// TIA Portal V17 export
// export: Created 2025-07-01T09:58:21.0344057Z, ExportSetting WithDefaults, DisplayName Totally Integrated Automation Portal, DisplayVersion V17 Update 8, DisplayName TIA Portal Openness, DisplayVersion V17 Update 8, DisplayName TIA Portal Version Control Interface, DisplayVersion V17, DisplayName SINAMICS Startdrive Advanced, DisplayVersion V17 SP2, DisplayName SINAMICS Startdrive G110M, G120, G120C, G120D, G120P, G115D, DisplayVersion V17 SP2, DisplayName SINAMICS Startdrive G130, G150, S120, S150, SINAMICS MV, S210, DisplayVersion V17 SP2, DisplayName STEP 7 Professional, DisplayVersion V17 Update 8, DisplayName SINUMERIK ONE STEP 7 Toolbox, DisplayVersion V17 Update 12, DisplayName SINUMERIK ONE PLC Basic Program Plus, DisplayVersion V17 Update 12, DisplayName SINUMERIK 840D sl STEP 7 Toolbox, DisplayVersion V17 Update 12, DisplayName STEP 7 Safety, DisplayVersion V17 Update 6, DisplayName WinCC Advanced, DisplayVersion V17 Update 8
FUNCTION_BLOCK "FB31_SPINDLE"   // FB31, LAD
{ S7_Optimized_Access := 'FALSE' }
AUTHOR : ETXETAR
VERSION : 1.0
// stored: AutoNumber false, IsIECCheckEnabled false, SetENOAutomatically false, UDAEnableTagReadback false
   VAR_INPUT
      OPTIONS_0 : Byte := 2#0000_0000;   // OPTIONS 0
      OPTIONS_1 : Byte := 2#0000_0000;   // OPTIONS 1
      SAFETY_BYPASS : Bool;   // MUST BE ALWAYS OFF, ACTIVATE ONLY FOR TEST
      OPTIMIZATION_BYPASS : Bool;   // MUST BE ALWAYS OFF, ACTIVATE ONLY FOR OPTIMIZATION TEST
      RPMS_REACHED : Bool;   // RPMS REACHED / N.O
      BELT_BROKEN : Bool;   // BELT BROKEN / N.C
      COOLING_SYS_IN_SERVICE : Bool;   // COOLING SYSTEM IN SERVICE
      MQL_HP_IN_SERVICE : Bool;   // MQL OR HP IN SERVICE
      TEMPERATURE_SENSOR : Word;   // TEMPERATURE SENSOR
      TEMPERATURE_SENSOR_PTC : Bool;   // TEMPERATURE SENSOR PTC
      VPM_READY : Bool;   // VOLTAGE PROTECTION MODULE READY
      ENABLE : Bool;   // ENABLE
      FEED_HOLD_COND : Bool;   // FEED HOLD CONDITION
      UNIT_SEQ_RUNNING : Bool;   // UNIT SEQUENCE RUNNING
      SAFE_ENABLED : Bool;   // SAFETY ENABLED
      TEST_STOP_INTERNAL_PULSES : Bool;   // TEST STOP INTERNAL PULSES
      FEED_OVERRIDE : Byte;   // FEED OVERRIDE
      SPINDLE_OVERRIDE : Byte;   // SPINDLE OVERRIDE
      HMI_SP_SELECTED : Bool;   // HMI SPINDLE SELECTED
      HMI_REQ_LINE : Bool;   // HMI REQUEST LINE
      CHANNEL_M3 : Bool;   // CHANNEL M3
      CHANNEL_M300 : Bool;   // CHANNEL M300
      M_VERIFY_CLAMP_F1 : Bool;   // M VERIFY CLAMPED FIXTURE 1
      M_VERIFY_CLAMP_F2 : Bool;   // M VERIFY CLAMPED FIXTURE 2
      SP_CLAMP : Bool;   // SPINDLE CLAMPING UNIT CLAMP
      SP_CLAMPED : Bool;   // SPINDLE CLAMPING UNIT CLAMPED
      SP_CLAMPED_WITH_TOOL : Bool;   // SPINDLE CLAMPING UNIT CLAMPED WITH TOOL
      HARDWARE_ENABLE : Bool;   // HARDWARE ENABLE
      TOOL_CHANGE_POS : Bool;   // TOOL CHANGE POSITION
      FIXTURE_1_PART_OK : Bool;   // FIXTURE 1 PART OK
      FIXTURE_2_PART_OK : Bool;   // FIXTURE 2 PART OK
      READ_POS : DWord;   // READ POSITION
      UNIT_ALARM : UInt;   // UNIT NUMBER MAX. NUMBER=10
      STATION_ALARM : UInt;   // STATION NUMBER MIN. NUMBER=0 MAX. NUMBER=4
      DESELECT_SPINDLE_STO : Bool;   // DESELECT SPINDLE STO
   END_VAR
   VAR_OUTPUT
      DELAYED_ENABLE : Bool;   // DELAYED ENABLE
      FEED_HOLD_CONDITIONS : Bool;   // FEED HOLD CONDITIONS
      FEED_HOLD_CONDITIONS_HMI : Bool;   // HMI FEED HOLD CONDITIONS
      SP_DESELECTED : Bool;   // SPINDLE DESELECTED
      SPEED_NOT_REACHED_ALARM : Bool;   // SPEED NOT REACHED ALARM
      BELT_BROKEN_ALARM : Bool;   // BELT BROKEN ALARM
      COOLING_ALARM : Bool;   // COOLING ALARM
      MQL_HP_ALARM : Bool;   // MQL HP ALARM
      HIGH_TEMP_ALARM : Bool;   // HIGH TEMPERATURE ALARM
      HIGH_TEMP_PTC_ALARM : Bool;   // HIGH TEMPERATURE PTC ALARM
      VPM_READY_ALARM : Bool;   // VPM READY ALARM
      HIGH_TEMP_PREALM : Bool;   // HIGH TEMPERATURE PREALARM
      SPINDLE_POS : Real;   // SPINDLE POSITION
      HMI_MOTION_EXECUTABILITY_LEFT : Bool;   // HMI MOTION EXECUTABILITY LEFT
      HMI_MOTION_EXECUTABILITY_RIGHT : Bool;   // HMI MOTION EXECUTABILITY RIGHT
      HMI_MOTION_END_POS_LEFT : Bool;   // HMI MOTION END POSITION LEFT
      HMI_MOTION_END_POS_RIGHT : Bool;   // HMI MOTION END POSITION RIGHT
   END_VAR
   VAR_IN_OUT
      SpindleDB : "LBP_typeAxisX";
   END_VAR
   VAR DB_SPECIFIC
      SP : "SPINDLE";
      SP_TEMPERATURE : Real;   // SPINDLE TEMPERATURE
      TEMP_MUL_VAL { S7_SetPoint := 'True'} : Real := 800.0;   // CONVERSION VALUE TO MUL THE INPUT
      TEMP_DIV_VAL { S7_SetPoint := 'True'} : Real := 16383.0;   // CONVERSION VALUE TO DIV THE MUL VALUE
      TEMP_SUB_VAL { S7_SetPoint := 'True'} : Real := 200.0;   // CONVERSION VALUE TO SUB TO THE SUB VALUE
      TEMP_PREALARM_VAL { S7_SetPoint := 'True'} : Real := 40.0;   // TEMPERATURE PREALARM VALUE
      TEMP_ALARM_VAL { S7_SetPoint := 'True'} : Real := 45.0;   // TEMPERATURE ALARM VALUE
      WARNING_GONE { S7_SetPoint := 'True'} : Bool;   // WARNING GONE
      TIMER_ENABLE_PULSE { S7_SetPoint := 'True'} : TOF_TIME;   // ENABLE PULSE TIMER
      TIMER_DELETE_DIST_TO_GO { S7_SetPoint := 'True'} : TON_TIME;   // DELETE DISTANCE TO GO TIMER
      TIMER_SPEED_NOT_REACHED { S7_SetPoint := 'True'} : TOF_TIME;   // SPEED NOT REACHED TIMER
      TIMER_BELT_BROKEN_ALARM { S7_SetPoint := 'True'} : TON_TIME;   // BELT BROKEN TIMER
      TIMER_MQL_HP_FAULT { S7_SetPoint := 'True'} : TON_TIME;   // MQL OR HP FAULT TIMER
      TIMER_COMMAND_JOG_PLUS { S7_SetPoint := 'True'} : TON_TIME;   // COMMAND JOG PLUS TIMER
   END_VAR
   VAR
      SAFETY_POSITIONS { S7_SetPoint := 'True'} : "FB33_SAFETY_POSITIONS";
   END_VAR
   VAR_TEMP
      INPUTS_MASK : Byte;   // INPUT MASK
      O_BYTE_0 : Struct   // OPTION BYTE 0
         MEASURING_SYSTEM_2 : Bool;   // MEASURING SYSTEM 2 OPTION / ALWAYS ON OR ALWAYS OFF
         BELT_BROKEN : Bool;   // BELT BROKEN OPTION
         COOLING : Bool;   // COOLING OPTION / ALWAYS ON OR ALWAYS OFF
         MQL_OR_HP : Bool;   // MQL OR HP OPTION / ALWAYS ON OR ALWAYS OFF
         ANALOG_TEMPERATURE_SENSOR : Bool;   // ANALOG TEMPERATURE SENSOR OPTION
         PTC_TEMP_SENSOR : Bool;   // PTC TEMPERATURE SENSOR OPTION
         TWIN_KESSLER_VPM_READY : Bool;   // TWIN KESSLER VPM READY OPTION
         MPP_SP_OVERRIDE : Bool;   // MPP SPINDLE OVERRIDE OPTION
      END_STRUCT;
      O_BYTE_1 : Struct   // OPTION BYTE 1
         SPARE_0 : Bool;   // SPARE OPTION / ALWAYS ON OR ALWAYS OFF
         SPARE_1 : Bool;   // SPARE OPTION
         SPARE_2 : Bool;   // SPARE OPTION / ALWAYS ON OR ALWAYS OFF
         SPARE_3 : Bool;   // SPARE OPTION / ALWAYS ON OR ALWAYS OFF
         SPARE_4 : Bool;   // SPARE OPTION
         SPARE_5 : Bool;   // SPARE OPTION
         SPARE_6 : Bool;   // SPARE OPTION
         SPARE_7 : Bool;   // SPARE OPTION
      END_STRUCT;
      TEMP_INPUT : DInt;   // TEMPERATURE INPUR SHIFTED
      TEMP_REAL : Real;   // TEMPERATURE IN REAL
      DB_NUMBER : DInt;   // DB NUMBER FOR ALARMS AND HELP DECODING
   END_VAR
   // TIMER_ENABLE_PULSE.PT := T#1s;
   // TIMER_DELETE_DIST_TO_GO.PT := T#20ms;
   // TIMER_SPEED_NOT_REACHED.PT := T#100ms;
   // TIMER_BELT_BROKEN_ALARM.PT := T#150ms;
   // TIMER_MQL_HP_FAULT.PT := T#50ms;
   // TIMER_COMMAND_JOG_PLUS.PT := T#100ms;
   VAR_TEMP   // added for the SCL form of the ladder/FBD networks
      _w1 : Bool;
      _w2 : Bool;
      _w3 : Bool;
      _w4 : Bool;
      _w5 : Bool;
      _w6 : Bool;
      _w7 : Bool;
      _w8 : Bool;
      _w9 : Bool;
      _w10 : Bool;
      _w11 : Bool;
   END_VAR
BEGIN

NETWORK
TITLE = READ INSTANCE DB
      L     DINO;
      +     10#800000;
      T     #DB_NUMBER;


REGION Network 2: OPTIONS
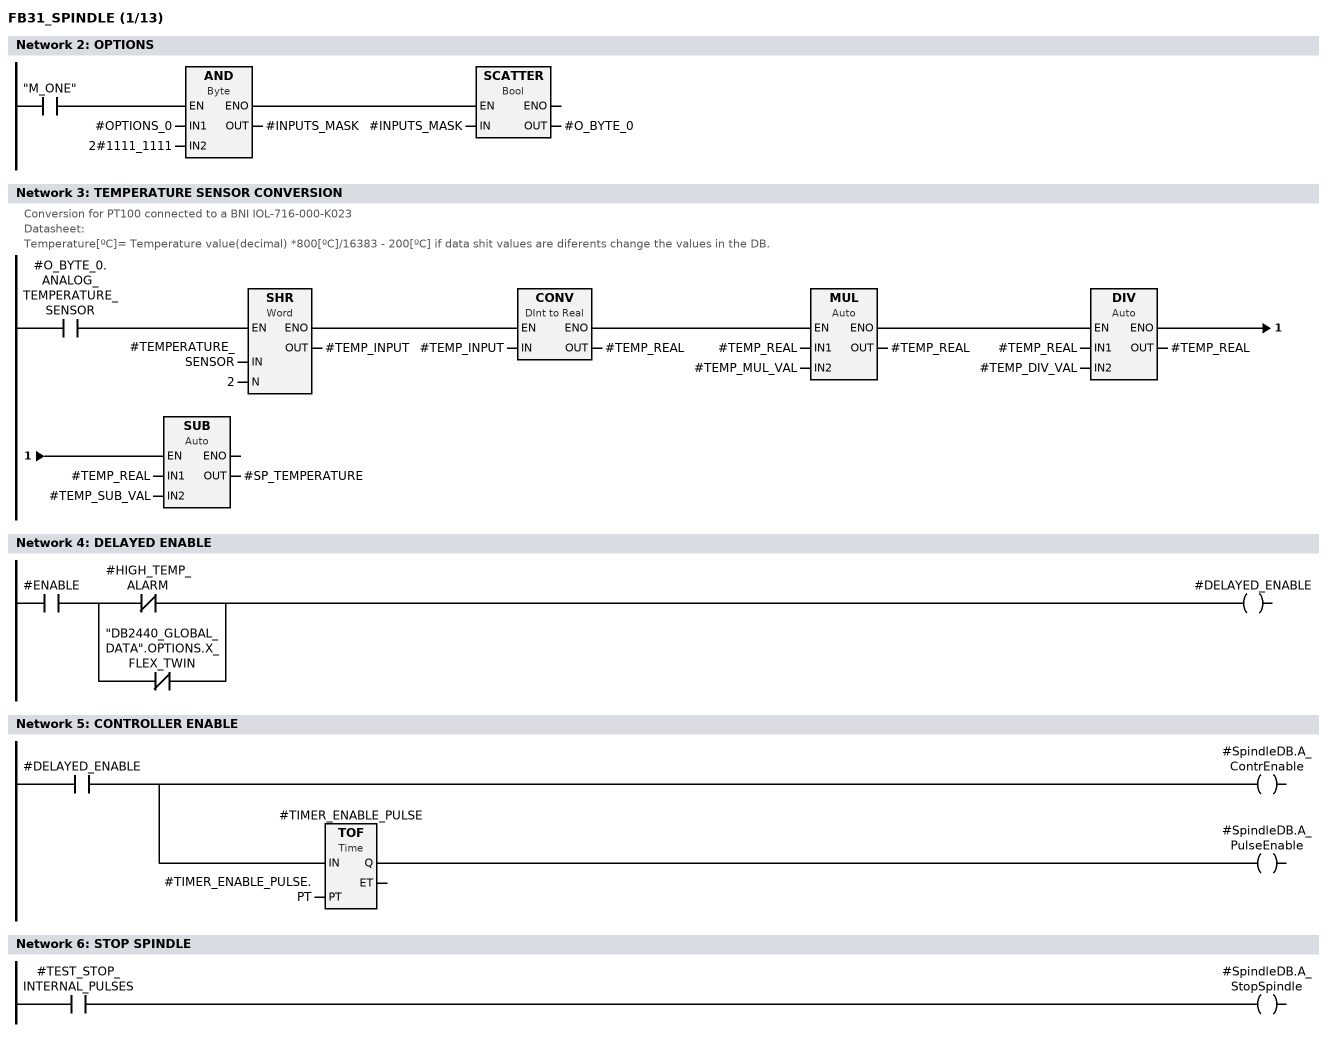
   RUNG wire#powerrail
      Contact( "M_ONE" )
      { S7_Templates := "SrcType := Byte"; S7_GenerateENO := "TRUE" } And(in1 := #OPTIONS_0, in2 := 2#1111_1111, out => #INPUTS_MASK)
      { S7_Templates := "[dest_type := Bool, src_type := Byte]" } SCATTER(IN := #INPUTS_MASK, OUT => #O_BYTE_0)
   END_RUNG
   // the same network as SCL:
   IF "M_ONE" THEN
       #INPUTS_MASK := #OPTIONS_0 AND 2#1111_1111;
       SCATTER(IN := #INPUTS_MASK, OUT => #O_BYTE_0);
   END_IF;
END_REGION

REGION Network 3: TEMPERATURE SENSOR CONVERSION
   // Conversion for PT100 connected to a BNI IOL-716-000-K023
   // 
   // Datasheet:
   // 
   //  Temperature[ºC]= Temperature value(decimal) *800[ºC]/16383 - 200[ºC] if data shit values are diferents change the values in the DB.
   RUNG wire#powerrail
      Contact( #O_BYTE_0.ANALOG_TEMPERATURE_SENSOR )
      { S7_Templates := "SrcType := Word" } Shr(in := #TEMPERATURE_SENSOR, n := 2, out => #TEMP_INPUT)
      { S7_Templates := "[SrcType := DInt, DestType := Real]" } Convert(in := #TEMP_INPUT, out => #TEMP_REAL)
      Mul(in1 := #TEMP_REAL, in2 := #TEMP_MUL_VAL, out => #TEMP_REAL)
      Div(in1 := #TEMP_REAL, in2 := #TEMP_DIV_VAL, out => #TEMP_REAL)
      Sub(in1 := #TEMP_REAL, in2 := #TEMP_SUB_VAL, out => #SP_TEMPERATURE)
   END_RUNG
   // the same network as SCL:
   IF #O_BYTE_0.ANALOG_TEMPERATURE_SENSOR THEN
       #TEMP_INPUT := SHR(IN := #TEMPERATURE_SENSOR, N := 2);
       #TEMP_REAL := DINT_TO_REAL(#TEMP_INPUT);
       #TEMP_REAL := #TEMP_REAL * #TEMP_MUL_VAL;
       #TEMP_REAL := #TEMP_REAL / #TEMP_DIV_VAL;
       #SP_TEMPERATURE := #TEMP_REAL - #TEMP_SUB_VAL;
   END_IF;
END_REGION

REGION Network 4: DELAYED ENABLE
   RUNG wire#powerrail
      Contact( #ENABLE )
      wire#w1
      I_Contact( #HIGH_TEMP_ALARM )
      wire#w2
      Coil( #DELAYED_ENABLE )
   END_RUNG
   RUNG wire#w1
      I_Contact( "DB2440_GLOBAL_DATA".OPTIONS.X_FLEX_TWIN )
   END_RUNG wire#w2
   // the same network as SCL:
   #DELAYED_ENABLE := #ENABLE AND (NOT #HIGH_TEMP_ALARM OR NOT "DB2440_GLOBAL_DATA".OPTIONS.X_FLEX_TWIN);
END_REGION

REGION Network 5: CONTROLLER ENABLE
   RUNG wire#powerrail
      Contact( #DELAYED_ENABLE )
      wire#w1
      Coil( #SpindleDB.A_ContrEnable )
   END_RUNG
   RUNG wire#w1
      { S7_Templates := "time_type := Time" } #TIMER_ENABLE_PULSE.TOF(pt := #TIMER_ENABLE_PULSE.PT, et =>)
      Coil( #SpindleDB.A_PulseEnable )
   END_RUNG
   // the same network as SCL:
   #SpindleDB.A_ContrEnable := #DELAYED_ENABLE;
   #TIMER_ENABLE_PULSE(IN := #DELAYED_ENABLE, PT := #TIMER_ENABLE_PULSE.PT);   // TOF
   #SpindleDB.A_PulseEnable := #TIMER_ENABLE_PULSE.Q;
END_REGION

REGION Network 6: STOP SPINDLE
   RUNG wire#powerrail
      Contact( #TEST_STOP_INTERNAL_PULSES )
      Coil( #SpindleDB.A_StopSpindle )
   END_RUNG
   // the same network as SCL:
   #SpindleDB.A_StopSpindle := #TEST_STOP_INTERNAL_PULSES;
END_REGION

REGION Network 7: DELETE DISTANCE TO GO / DELETE S VALUE
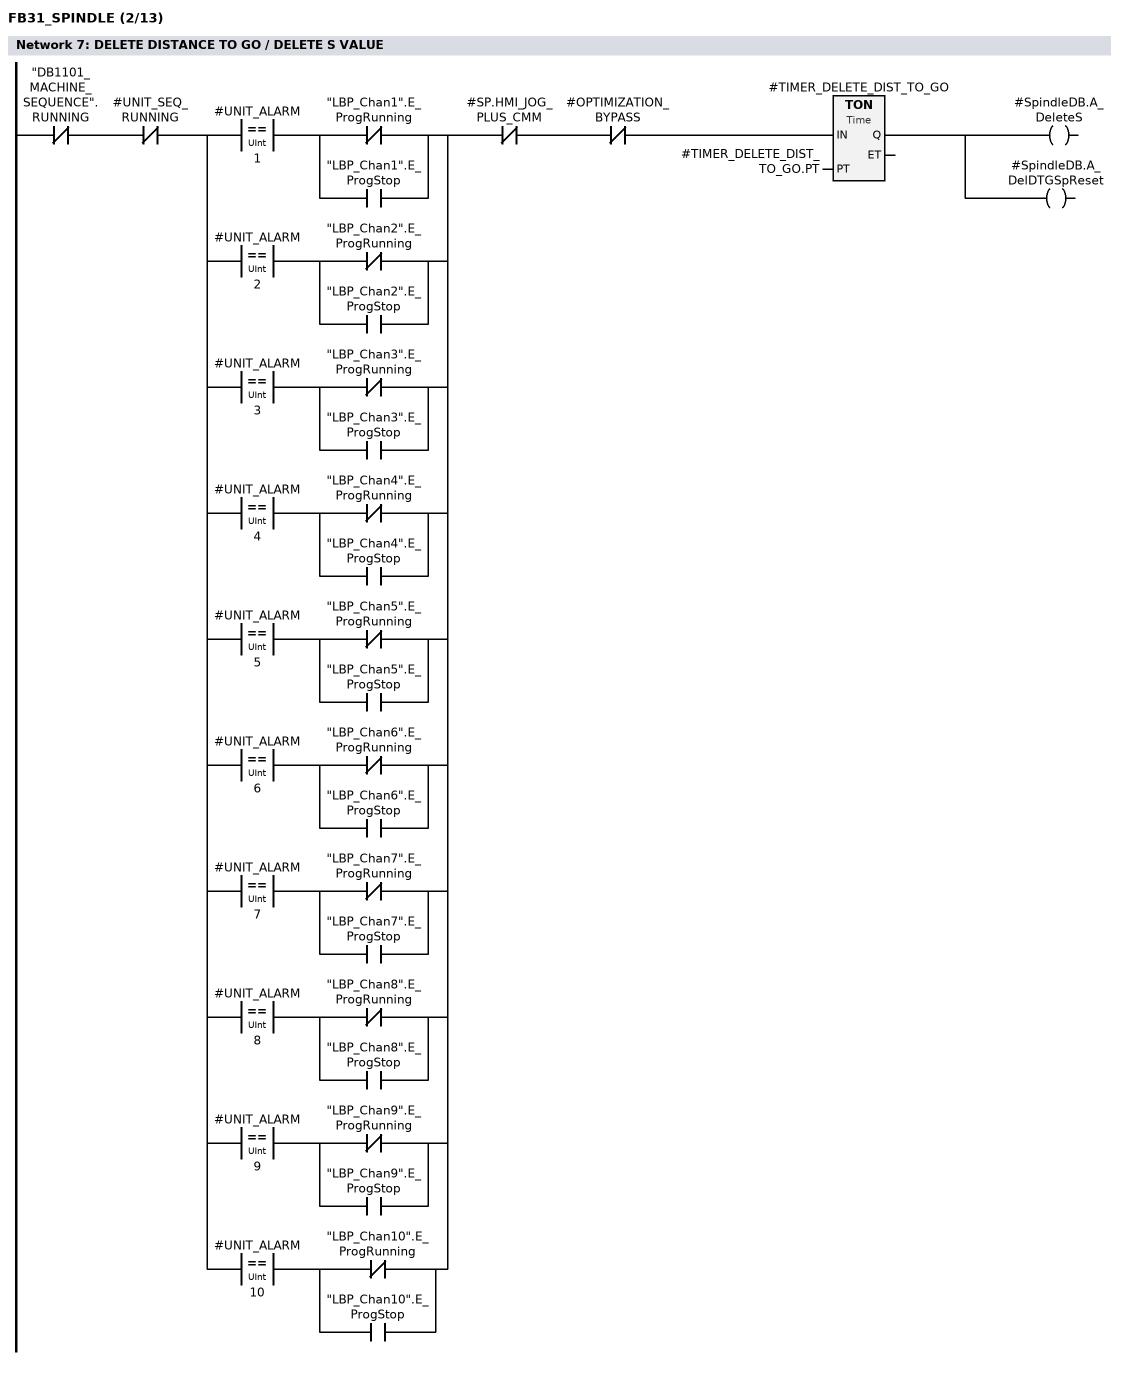
   RUNG wire#powerrail
      I_Contact( "DB1101_MACHINE_SEQUENCE".RUNNING )
      I_Contact( #UNIT_SEQ_RUNNING )
      wire#w1
      { S7_Templates := "SrcType := UInt" } EQ_Contact(in1 := #UNIT_ALARM, in2 := 1)
      wire#w2
      I_Contact( "LBP_Chan1".E_ProgRunning )
      wire#w3
      I_Contact( #SP.HMI_JOG_PLUS_CMM )
      I_Contact( #OPTIMIZATION_BYPASS )
      { S7_Templates := "time_type := Time" } #TIMER_DELETE_DIST_TO_GO.TON(pt := #TIMER_DELETE_DIST_TO_GO.PT, et =>)
      wire#w13
      Coil( #SpindleDB.A_DeleteS )
   END_RUNG
   RUNG wire#w2
      Contact( "LBP_Chan1".E_ProgStop )
   END_RUNG wire#w3
   RUNG wire#w1
      { S7_Templates := "SrcType := UInt" } EQ_Contact(in1 := #UNIT_ALARM, in2 := 2)
      wire#w4
      I_Contact( "LBP_Chan2".E_ProgRunning )
   END_RUNG wire#w3
   RUNG wire#w4
      Contact( "LBP_Chan2".E_ProgStop )
   END_RUNG wire#w3
   RUNG wire#w1
      { S7_Templates := "SrcType := UInt" } EQ_Contact(in1 := #UNIT_ALARM, in2 := 3)
      wire#w5
      I_Contact( "LBP_Chan3".E_ProgRunning )
   END_RUNG wire#w3
   RUNG wire#w5
      Contact( "LBP_Chan3".E_ProgStop )
   END_RUNG wire#w3
   RUNG wire#w1
      { S7_Templates := "SrcType := UInt" } EQ_Contact(in1 := #UNIT_ALARM, in2 := 4)
      wire#w6
      I_Contact( "LBP_Chan4".E_ProgRunning )
   END_RUNG wire#w3
   RUNG wire#w6
      Contact( "LBP_Chan4".E_ProgStop )
   END_RUNG wire#w3
   RUNG wire#w1
      { S7_Templates := "SrcType := UInt" } EQ_Contact(in1 := #UNIT_ALARM, in2 := 5)
      wire#w7
      I_Contact( "LBP_Chan5".E_ProgRunning )
   END_RUNG wire#w3
   RUNG wire#w7
      Contact( "LBP_Chan5".E_ProgStop )
   END_RUNG wire#w3
   RUNG wire#w1
      { S7_Templates := "SrcType := UInt" } EQ_Contact(in1 := #UNIT_ALARM, in2 := 6)
      wire#w8
      I_Contact( "LBP_Chan6".E_ProgRunning )
   END_RUNG wire#w3
   RUNG wire#w8
      Contact( "LBP_Chan6".E_ProgStop )
   END_RUNG wire#w3
   RUNG wire#w1
      { S7_Templates := "SrcType := UInt" } EQ_Contact(in1 := #UNIT_ALARM, in2 := 7)
      wire#w9
      I_Contact( "LBP_Chan7".E_ProgRunning )
   END_RUNG wire#w3
   RUNG wire#w9
      Contact( "LBP_Chan7".E_ProgStop )
   END_RUNG wire#w3
   RUNG wire#w1
      { S7_Templates := "SrcType := UInt" } EQ_Contact(in1 := #UNIT_ALARM, in2 := 8)
      wire#w10
      I_Contact( "LBP_Chan8".E_ProgRunning )
   END_RUNG wire#w3
   RUNG wire#w10
      Contact( "LBP_Chan8".E_ProgStop )
   END_RUNG wire#w3
   RUNG wire#w1
      { S7_Templates := "SrcType := UInt" } EQ_Contact(in1 := #UNIT_ALARM, in2 := 9)
      wire#w11
      I_Contact( "LBP_Chan9".E_ProgRunning )
   END_RUNG wire#w3
   RUNG wire#w11
      Contact( "LBP_Chan9".E_ProgStop )
   END_RUNG wire#w3
   RUNG wire#w1
      { S7_Templates := "SrcType := UInt" } EQ_Contact(in1 := #UNIT_ALARM, in2 := 10)
      wire#w12
      I_Contact( "LBP_Chan10".E_ProgRunning )
   END_RUNG wire#w3
   RUNG wire#w12
      Contact( "LBP_Chan10".E_ProgStop )
   END_RUNG wire#w3
   RUNG wire#w13
      Coil( #SpindleDB.A_DelDTGSpReset )
   END_RUNG
   // the same network as SCL:
   #TIMER_DELETE_DIST_TO_GO(IN := NOT "DB1101_MACHINE_SEQUENCE".RUNNING AND NOT #UNIT_SEQ_RUNNING AND (((#UNIT_ALARM = 1) AND (NOT "LBP_Chan1".E_ProgRunning OR "LBP_Chan1".E_ProgStop)) OR ((#UNIT_ALARM = 2) AND (NOT "LBP_Chan2".E_ProgRunning OR "LBP_Chan2".E_ProgStop)) OR ((#UNIT_ALARM = 3) AND (NOT "LBP_Chan3".E_ProgRunning OR "LBP_Chan3".E_ProgStop)) OR ((#UNIT_ALARM = 4) AND (NOT "LBP_Chan4".E_ProgRunning OR "LBP_Chan4".E_ProgStop)) OR ((#UNIT_ALARM = 5) AND (NOT "LBP_Chan5".E_ProgRunning OR "LBP_Chan5".E_ProgStop)) OR ((#UNIT_ALARM = 6) AND (NOT "LBP_Chan6".E_ProgRunning OR "LBP_Chan6".E_ProgStop)) OR ((#UNIT_ALARM = 7) AND (NOT "LBP_Chan7".E_ProgRunning OR "LBP_Chan7".E_ProgStop)) OR ((#UNIT_ALARM = 8) AND (NOT "LBP_Chan8".E_ProgRunning OR "LBP_Chan8".E_ProgStop)) OR ((#UNIT_ALARM = 9) AND (NOT "LBP_Chan9".E_ProgRunning OR "LBP_Chan9".E_ProgStop)) OR ((#UNIT_ALARM = 10) AND (NOT "LBP_Chan10".E_ProgRunning OR "LBP_Chan10".E_ProgStop))) AND NOT #SP.HMI_JOG_PLUS_CMM AND NOT #OPTIMIZATION_BYPASS,   // TON
                           PT := #TIMER_DELETE_DIST_TO_GO.PT);
   #SpindleDB.A_DeleteS := #TIMER_DELETE_DIST_TO_GO.Q;
   #SpindleDB.A_DelDTGSpReset := #TIMER_DELETE_DIST_TO_GO.Q;
END_REGION

REGION Network 8: POSITION MEASURING SYTEM
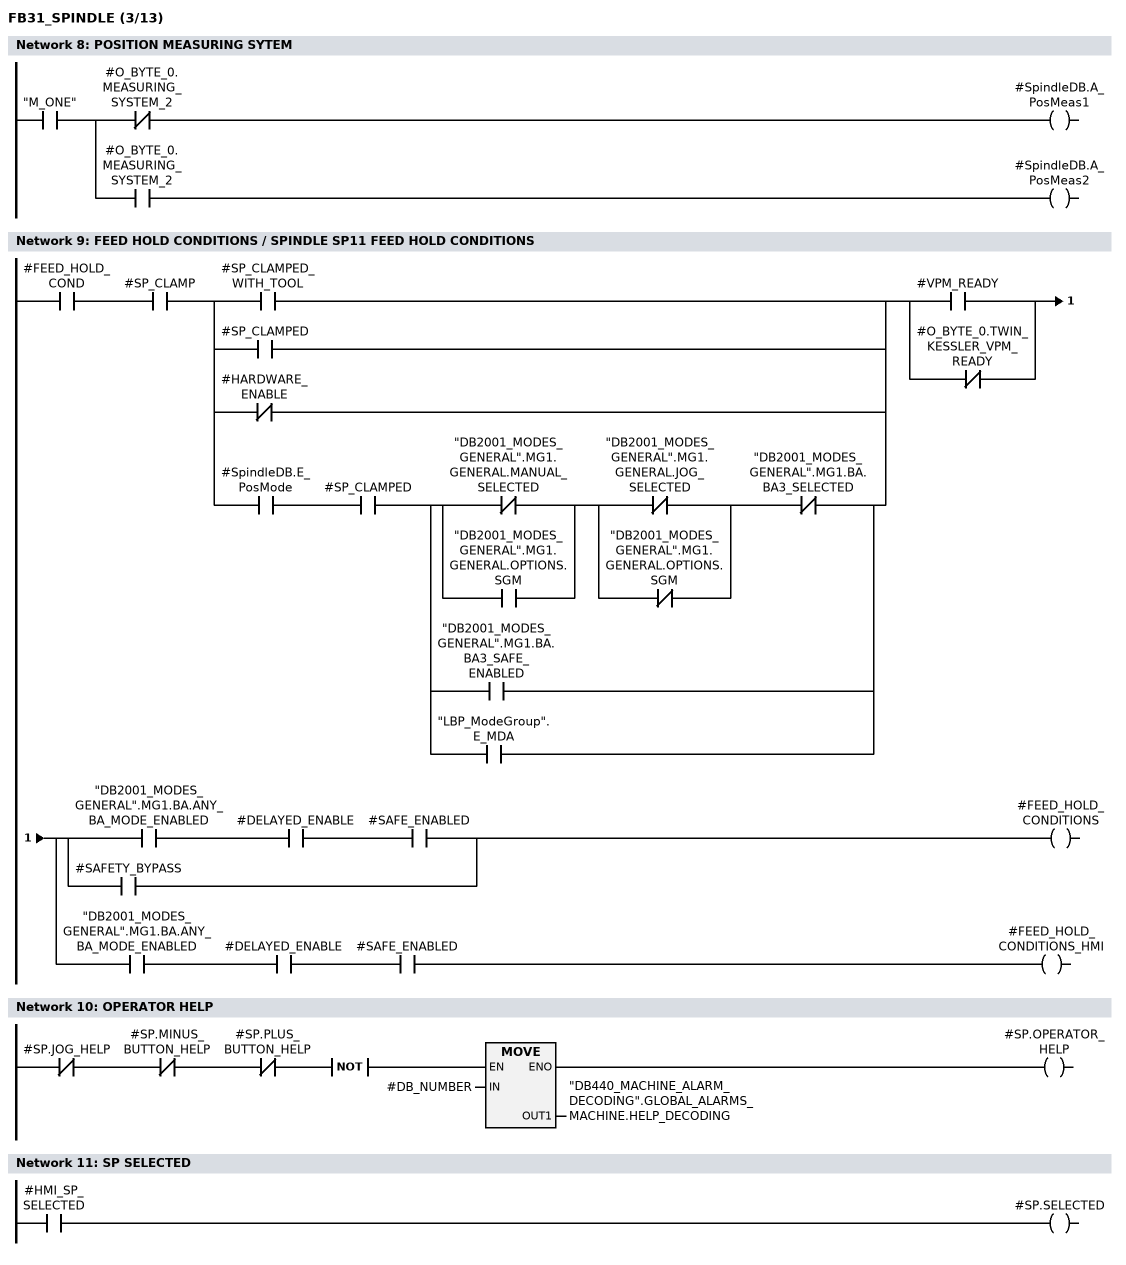
   RUNG wire#powerrail
      Contact( "M_ONE" )
      wire#w1
      I_Contact( #O_BYTE_0.MEASURING_SYSTEM_2 )
      Coil( #SpindleDB.A_PosMeas1 )
   END_RUNG
   RUNG wire#w1
      Contact( #O_BYTE_0.MEASURING_SYSTEM_2 )
      Coil( #SpindleDB.A_PosMeas2 )
   END_RUNG
   // the same network as SCL:
   #SpindleDB.A_PosMeas1 := "M_ONE" AND NOT #O_BYTE_0.MEASURING_SYSTEM_2;
   #SpindleDB.A_PosMeas2 := "M_ONE" AND #O_BYTE_0.MEASURING_SYSTEM_2;
END_REGION

REGION Network 9: FEED HOLD CONDITIONS / SPINDLE SP11 FEED HOLD CONDITIONS
   RUNG wire#powerrail
      Contact( #FEED_HOLD_COND )
      Contact( #SP_CLAMP )
      wire#w1
      Contact( #SP_CLAMPED_WITH_TOOL )
      wire#w2
      Contact( #VPM_READY )
      wire#w6
      Contact( "DB2001_MODES_GENERAL".MG1.BA.ANY_BA_MODE_ENABLED )
      Contact( #DELAYED_ENABLE )
      Contact( #SAFE_ENABLED )
      wire#w7
      Coil( #FEED_HOLD_CONDITIONS )
   END_RUNG
   RUNG wire#w1
      Contact( #SP_CLAMPED )
   END_RUNG wire#w2
   RUNG wire#w1
      I_Contact( #HARDWARE_ENABLE )
   END_RUNG wire#w2
   RUNG wire#w1
      Contact( #SpindleDB.E_PosMode )
      Contact( #SP_CLAMPED )
      wire#w3
      I_Contact( "DB2001_MODES_GENERAL".MG1.GENERAL.MANUAL_SELECTED )
      wire#w4
      I_Contact( "DB2001_MODES_GENERAL".MG1.GENERAL.JOG_SELECTED )
      wire#w5
      I_Contact( "DB2001_MODES_GENERAL".MG1.BA.BA3_SELECTED )
   END_RUNG wire#w2
   RUNG wire#w3
      Contact( "DB2001_MODES_GENERAL".MG1.GENERAL.OPTIONS.SGM )
   END_RUNG wire#w4
   RUNG wire#w4
      I_Contact( "DB2001_MODES_GENERAL".MG1.GENERAL.OPTIONS.SGM )
   END_RUNG wire#w5
   RUNG wire#w3
      Contact( "DB2001_MODES_GENERAL".MG1.BA.BA3_SAFE_ENABLED )
   END_RUNG wire#w2
   RUNG wire#w3
      Contact( "LBP_ModeGroup".E_MDA )
   END_RUNG wire#w2
   RUNG wire#w2
      I_Contact( #O_BYTE_0.TWIN_KESSLER_VPM_READY )
   END_RUNG wire#w6
   RUNG wire#w6
      Contact( #SAFETY_BYPASS )
   END_RUNG wire#w7
   RUNG wire#w6
      Contact( "DB2001_MODES_GENERAL".MG1.BA.ANY_BA_MODE_ENABLED )
      Contact( #DELAYED_ENABLE )
      Contact( #SAFE_ENABLED )
      Coil( #FEED_HOLD_CONDITIONS_HMI )
   END_RUNG
   // the same network as SCL:
   #_w1 := #FEED_HOLD_COND AND #SP_CLAMP AND (#SP_CLAMPED_WITH_TOOL OR #SP_CLAMPED OR NOT #HARDWARE_ENABLE OR (#SpindleDB.E_PosMode AND #SP_CLAMPED AND (((NOT "DB2001_MODES_GENERAL".MG1.GENERAL.MANUAL_SELECTED OR "DB2001_MODES_GENERAL".MG1.GENERAL.OPTIONS.SGM) AND (NOT "DB2001_MODES_GENERAL".MG1.GENERAL.JOG_SELECTED OR NOT "DB2001_MODES_GENERAL".MG1.GENERAL.OPTIONS.SGM) AND NOT "DB2001_MODES_GENERAL".MG1.BA.BA3_SELECTED) OR "DB2001_MODES_GENERAL".MG1.BA.BA3_SAFE_ENABLED OR "LBP_ModeGroup".E_MDA))) AND (#VPM_READY OR NOT #O_BYTE_0.TWIN_KESSLER_VPM_READY);
   #FEED_HOLD_CONDITIONS := #_w1 AND (("DB2001_MODES_GENERAL".MG1.BA.ANY_BA_MODE_ENABLED AND #DELAYED_ENABLE AND #SAFE_ENABLED) OR #SAFETY_BYPASS);
   #FEED_HOLD_CONDITIONS_HMI := #_w1 AND "DB2001_MODES_GENERAL".MG1.BA.ANY_BA_MODE_ENABLED AND #DELAYED_ENABLE AND #SAFE_ENABLED;
END_REGION

REGION Network 10: OPERATOR HELP
   RUNG wire#powerrail
      I_Contact( #SP.JOG_HELP )
      I_Contact( #SP.MINUS_BUTTON_HELP )
      I_Contact( #SP.PLUS_BUTTON_HELP )
      Not()
      { S7_GenerateENO := "TRUE" } Move(in := #DB_NUMBER, out1 => "DB440_MACHINE_ALARM_DECODING".GLOBAL_ALARMS_MACHINE.HELP_DECODING)
      Coil( #SP.OPERATOR_HELP )
   END_RUNG
   // the same network as SCL:
   // ENO of a box is taken as its EN; it also drops when the box reports an error
   #_w1 := NOT (NOT #SP.JOG_HELP AND NOT #SP.MINUS_BUTTON_HELP AND NOT #SP.PLUS_BUTTON_HELP);
   IF #_w1 THEN "DB440_MACHINE_ALARM_DECODING".GLOBAL_ALARMS_MACHINE.HELP_DECODING := #DB_NUMBER; END_IF;
   #SP.OPERATOR_HELP := #_w1;
END_REGION

REGION Network 11: SP SELECTED
   RUNG wire#powerrail
      Contact( #HMI_SP_SELECTED )
      Coil( #SP.SELECTED )
   END_RUNG
   // the same network as SCL:
   #SP.SELECTED := #HMI_SP_SELECTED;
END_REGION

REGION Network 12: SP DESELECTED
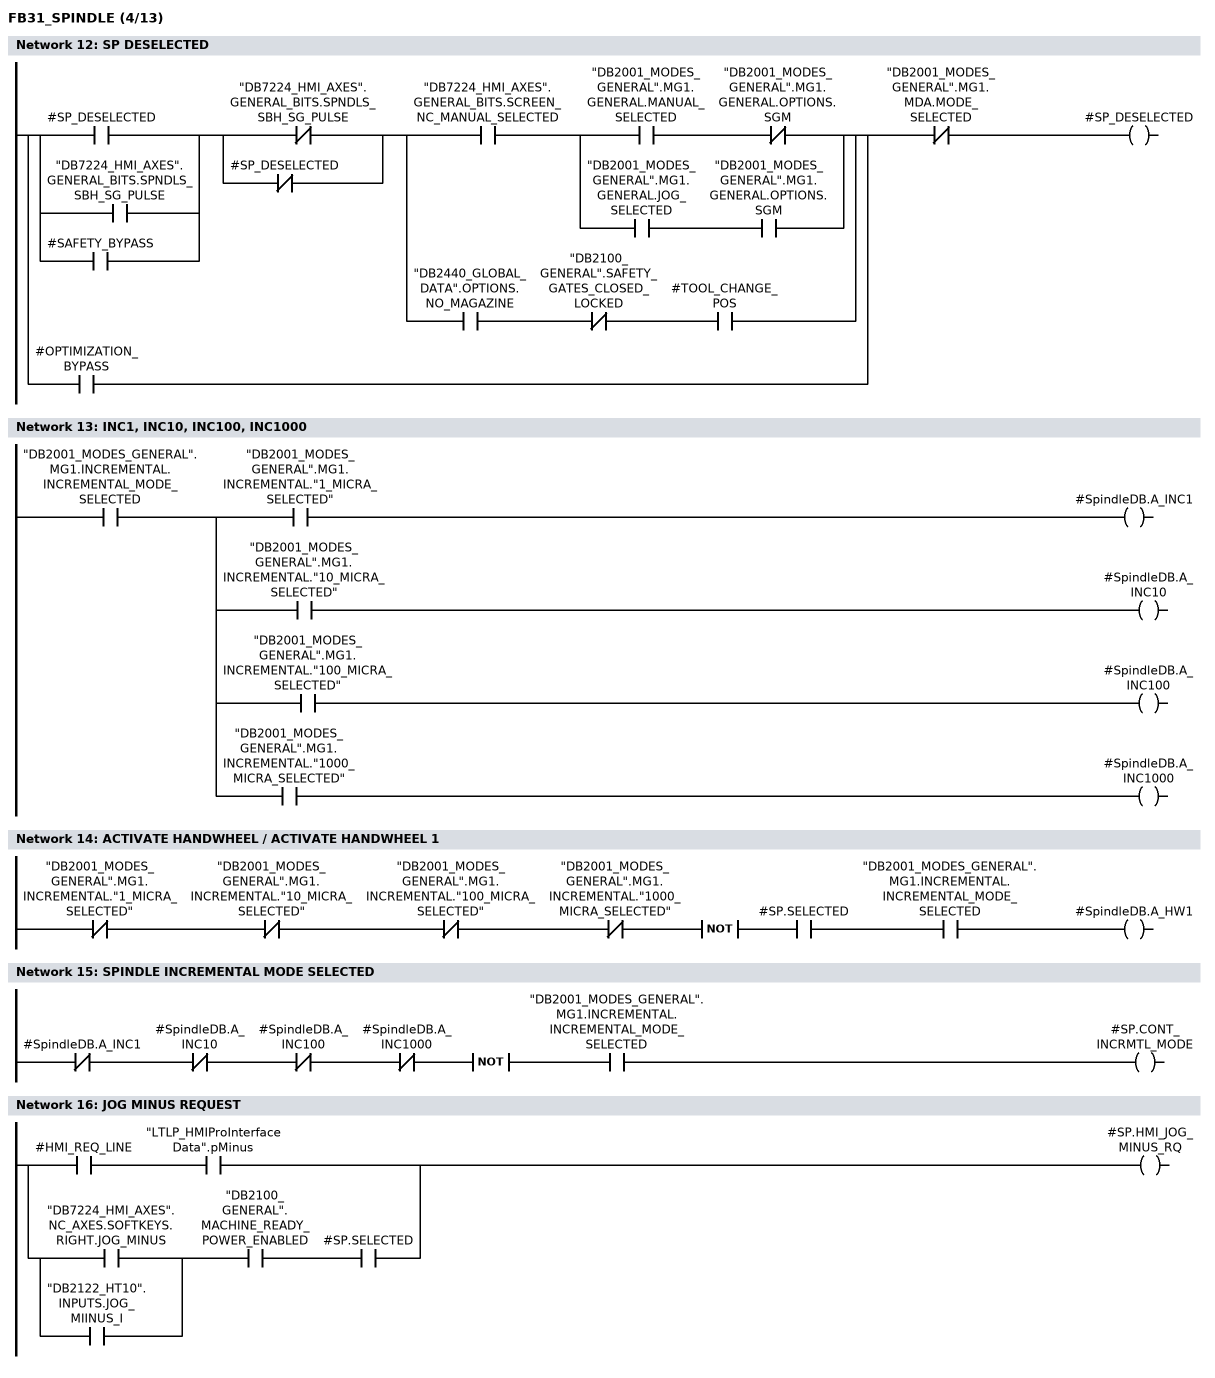
   RUNG wire#powerrail
      Contact( #SP_DESELECTED )
      wire#w1
      I_Contact( "DB7224_HMI_AXES".GENERAL_BITS.SPNDLS_SBH_SG_PULSE )
      wire#w2
      Contact( "DB7224_HMI_AXES".GENERAL_BITS.SCREEN_NC_MANUAL_SELECTED )
      wire#w3
      Contact( "DB2001_MODES_GENERAL".MG1.GENERAL.MANUAL_SELECTED )
      I_Contact( "DB2001_MODES_GENERAL".MG1.GENERAL.OPTIONS.SGM )
      wire#w4
      I_Contact( "DB2001_MODES_GENERAL".MG1.MDA.MODE_SELECTED )
      Coil( #SP_DESELECTED )
   END_RUNG
   RUNG wire#powerrail
      Contact( "DB7224_HMI_AXES".GENERAL_BITS.SPNDLS_SBH_SG_PULSE )
   END_RUNG wire#w1
   RUNG wire#powerrail
      Contact( #SAFETY_BYPASS )
   END_RUNG wire#w1
   RUNG wire#w1
      I_Contact( #SP_DESELECTED )
   END_RUNG wire#w2
   RUNG wire#w3
      Contact( "DB2001_MODES_GENERAL".MG1.GENERAL.JOG_SELECTED )
      Contact( "DB2001_MODES_GENERAL".MG1.GENERAL.OPTIONS.SGM )
   END_RUNG wire#w4
   RUNG wire#w2
      Contact( "DB2440_GLOBAL_DATA".OPTIONS.NO_MAGAZINE )
      I_Contact( "DB2100_GENERAL".SAFETY_GATES_CLOSED_LOCKED )
      Contact( #TOOL_CHANGE_POS )
   END_RUNG wire#w4
   RUNG wire#powerrail
      Contact( #OPTIMIZATION_BYPASS )
   END_RUNG wire#w4
   // the same network as SCL:
   #SP_DESELECTED := (((#SP_DESELECTED OR "DB7224_HMI_AXES".GENERAL_BITS.SPNDLS_SBH_SG_PULSE OR #SAFETY_BYPASS) AND (NOT "DB7224_HMI_AXES".GENERAL_BITS.SPNDLS_SBH_SG_PULSE OR NOT #SP_DESELECTED) AND (("DB7224_HMI_AXES".GENERAL_BITS.SCREEN_NC_MANUAL_SELECTED AND (("DB2001_MODES_GENERAL".MG1.GENERAL.MANUAL_SELECTED AND NOT "DB2001_MODES_GENERAL".MG1.GENERAL.OPTIONS.SGM) OR ("DB2001_MODES_GENERAL".MG1.GENERAL.JOG_SELECTED AND "DB2001_MODES_GENERAL".MG1.GENERAL.OPTIONS.SGM))) OR ("DB2440_GLOBAL_DATA".OPTIONS.NO_MAGAZINE AND NOT "DB2100_GENERAL".SAFETY_GATES_CLOSED_LOCKED AND #TOOL_CHANGE_POS))) OR #OPTIMIZATION_BYPASS) AND NOT "DB2001_MODES_GENERAL".MG1.MDA.MODE_SELECTED;
END_REGION

REGION Network 13: INC1, INC10, INC100, INC1000
   RUNG wire#powerrail
      Contact( "DB2001_MODES_GENERAL".MG1.INCREMENTAL.INCREMENTAL_MODE_SELECTED )
      wire#w1
      Contact( "DB2001_MODES_GENERAL".MG1.INCREMENTAL."1_MICRA_SELECTED" )
      Coil( #SpindleDB.A_INC1 )
   END_RUNG
   RUNG wire#w1
      Contact( "DB2001_MODES_GENERAL".MG1.INCREMENTAL."10_MICRA_SELECTED" )
      Coil( #SpindleDB.A_INC10 )
   END_RUNG
   RUNG wire#w1
      Contact( "DB2001_MODES_GENERAL".MG1.INCREMENTAL."100_MICRA_SELECTED" )
      Coil( #SpindleDB.A_INC100 )
   END_RUNG
   RUNG wire#w1
      Contact( "DB2001_MODES_GENERAL".MG1.INCREMENTAL."1000_MICRA_SELECTED" )
      Coil( #SpindleDB.A_INC1000 )
   END_RUNG
   // the same network as SCL:
   #SpindleDB.A_INC1 := "DB2001_MODES_GENERAL".MG1.INCREMENTAL.INCREMENTAL_MODE_SELECTED AND "DB2001_MODES_GENERAL".MG1.INCREMENTAL."1_MICRA_SELECTED";
   #SpindleDB.A_INC10 := "DB2001_MODES_GENERAL".MG1.INCREMENTAL.INCREMENTAL_MODE_SELECTED AND "DB2001_MODES_GENERAL".MG1.INCREMENTAL."10_MICRA_SELECTED";
   #SpindleDB.A_INC100 := "DB2001_MODES_GENERAL".MG1.INCREMENTAL.INCREMENTAL_MODE_SELECTED AND "DB2001_MODES_GENERAL".MG1.INCREMENTAL."100_MICRA_SELECTED";
   #SpindleDB.A_INC1000 := "DB2001_MODES_GENERAL".MG1.INCREMENTAL.INCREMENTAL_MODE_SELECTED AND "DB2001_MODES_GENERAL".MG1.INCREMENTAL."1000_MICRA_SELECTED";
END_REGION

REGION Network 14: ACTIVATE HANDWHEEL / ACTIVATE HANDWHEEL 1
   RUNG wire#powerrail
      I_Contact( "DB2001_MODES_GENERAL".MG1.INCREMENTAL."1_MICRA_SELECTED" )
      I_Contact( "DB2001_MODES_GENERAL".MG1.INCREMENTAL."10_MICRA_SELECTED" )
      I_Contact( "DB2001_MODES_GENERAL".MG1.INCREMENTAL."100_MICRA_SELECTED" )
      I_Contact( "DB2001_MODES_GENERAL".MG1.INCREMENTAL."1000_MICRA_SELECTED" )
      Not()
      Contact( #SP.SELECTED )
      Contact( "DB2001_MODES_GENERAL".MG1.INCREMENTAL.INCREMENTAL_MODE_SELECTED )
      Coil( #SpindleDB.A_HW1 )
   END_RUNG
   // the same network as SCL:
   #SpindleDB.A_HW1 := NOT (NOT "DB2001_MODES_GENERAL".MG1.INCREMENTAL."1_MICRA_SELECTED" AND NOT "DB2001_MODES_GENERAL".MG1.INCREMENTAL."10_MICRA_SELECTED" AND NOT "DB2001_MODES_GENERAL".MG1.INCREMENTAL."100_MICRA_SELECTED" AND NOT "DB2001_MODES_GENERAL".MG1.INCREMENTAL."1000_MICRA_SELECTED") AND #SP.SELECTED AND "DB2001_MODES_GENERAL".MG1.INCREMENTAL.INCREMENTAL_MODE_SELECTED;
END_REGION

REGION Network 15: SPINDLE INCREMENTAL MODE SELECTED
   RUNG wire#powerrail
      I_Contact( #SpindleDB.A_INC1 )
      I_Contact( #SpindleDB.A_INC10 )
      I_Contact( #SpindleDB.A_INC100 )
      I_Contact( #SpindleDB.A_INC1000 )
      Not()
      Contact( "DB2001_MODES_GENERAL".MG1.INCREMENTAL.INCREMENTAL_MODE_SELECTED )
      Coil( #SP.CONT_INCRMTL_MODE )
   END_RUNG
   // the same network as SCL:
   #SP.CONT_INCRMTL_MODE := NOT (NOT #SpindleDB.A_INC1 AND NOT #SpindleDB.A_INC10 AND NOT #SpindleDB.A_INC100 AND NOT #SpindleDB.A_INC1000) AND "DB2001_MODES_GENERAL".MG1.INCREMENTAL.INCREMENTAL_MODE_SELECTED;
END_REGION

REGION Network 16: JOG MINUS REQUEST
   RUNG wire#powerrail
      Contact( #HMI_REQ_LINE )
      Contact( "LTLP_HMIProInterfaceData".pMinus )
      wire#w1
      Coil( #SP.HMI_JOG_MINUS_RQ )
   END_RUNG
   RUNG wire#powerrail
      Contact( "DB7224_HMI_AXES".NC_AXES.SOFTKEYS.RIGHT.JOG_MINUS )
      wire#w2
      Contact( "DB2100_GENERAL".MACHINE_READY_POWER_ENABLED )
      Contact( #SP.SELECTED )
   END_RUNG wire#w1
   RUNG wire#powerrail
      Contact( "DB2122_HT10".INPUTS.JOG_MIINUS_I )
   END_RUNG wire#w2
   // the same network as SCL:
   #SP.HMI_JOG_MINUS_RQ := (#HMI_REQ_LINE AND "LTLP_HMIProInterfaceData".pMinus) OR (("DB7224_HMI_AXES".NC_AXES.SOFTKEYS.RIGHT.JOG_MINUS OR "DB2122_HT10".INPUTS.JOG_MIINUS_I) AND "DB2100_GENERAL".MACHINE_READY_POWER_ENABLED AND #SP.SELECTED);
END_REGION

REGION Network 17: JOG MINUS COMMAND
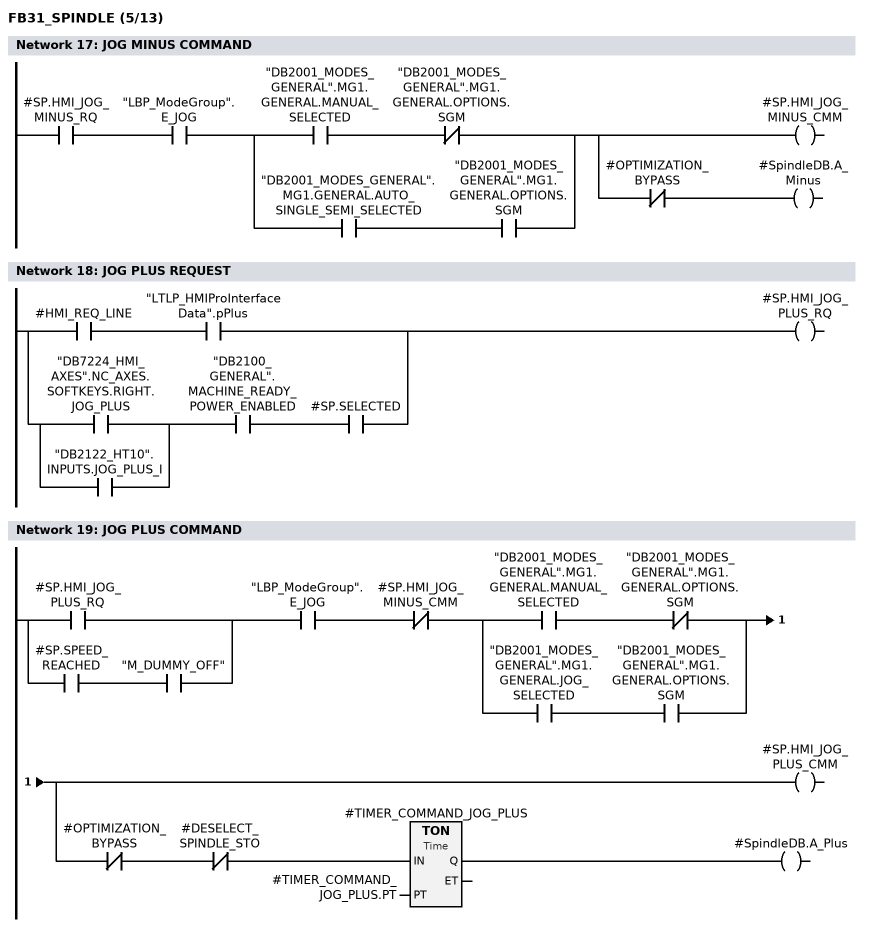
   RUNG wire#powerrail
      Contact( #SP.HMI_JOG_MINUS_RQ )
      Contact( "LBP_ModeGroup".E_JOG )
      wire#w1
      Contact( "DB2001_MODES_GENERAL".MG1.GENERAL.MANUAL_SELECTED )
      I_Contact( "DB2001_MODES_GENERAL".MG1.GENERAL.OPTIONS.SGM )
      wire#w2
      Coil( #SP.HMI_JOG_MINUS_CMM )
   END_RUNG
   RUNG wire#w1
      Contact( "DB2001_MODES_GENERAL".MG1.GENERAL.AUTO_SINGLE_SEMI_SELECTED )
      Contact( "DB2001_MODES_GENERAL".MG1.GENERAL.OPTIONS.SGM )
   END_RUNG wire#w2
   RUNG wire#w2
      I_Contact( #OPTIMIZATION_BYPASS )
      Coil( #SpindleDB.A_Minus )
   END_RUNG
   // the same network as SCL:
   #SP.HMI_JOG_MINUS_CMM := #SP.HMI_JOG_MINUS_RQ AND "LBP_ModeGroup".E_JOG AND (("DB2001_MODES_GENERAL".MG1.GENERAL.MANUAL_SELECTED AND NOT "DB2001_MODES_GENERAL".MG1.GENERAL.OPTIONS.SGM) OR ("DB2001_MODES_GENERAL".MG1.GENERAL.AUTO_SINGLE_SEMI_SELECTED AND "DB2001_MODES_GENERAL".MG1.GENERAL.OPTIONS.SGM));
   #SpindleDB.A_Minus := #SP.HMI_JOG_MINUS_CMM AND NOT #OPTIMIZATION_BYPASS;
END_REGION

REGION Network 18: JOG PLUS REQUEST
   RUNG wire#powerrail
      Contact( #HMI_REQ_LINE )
      Contact( "LTLP_HMIProInterfaceData".pPlus )
      wire#w1
      Coil( #SP.HMI_JOG_PLUS_RQ )
   END_RUNG
   RUNG wire#powerrail
      Contact( "DB7224_HMI_AXES".NC_AXES.SOFTKEYS.RIGHT.JOG_PLUS )
      wire#w2
      Contact( "DB2100_GENERAL".MACHINE_READY_POWER_ENABLED )
      Contact( #SP.SELECTED )
   END_RUNG wire#w1
   RUNG wire#powerrail
      Contact( "DB2122_HT10".INPUTS.JOG_PLUS_I )
   END_RUNG wire#w2
   // the same network as SCL:
   #SP.HMI_JOG_PLUS_RQ := (#HMI_REQ_LINE AND "LTLP_HMIProInterfaceData".pPlus) OR (("DB7224_HMI_AXES".NC_AXES.SOFTKEYS.RIGHT.JOG_PLUS OR "DB2122_HT10".INPUTS.JOG_PLUS_I) AND "DB2100_GENERAL".MACHINE_READY_POWER_ENABLED AND #SP.SELECTED);
END_REGION

REGION Network 19: JOG PLUS COMMAND
   RUNG wire#powerrail
      Contact( #SP.HMI_JOG_PLUS_RQ )
      wire#w1
      Contact( "LBP_ModeGroup".E_JOG )
      I_Contact( #SP.HMI_JOG_MINUS_CMM )
      wire#w2
      Contact( "DB2001_MODES_GENERAL".MG1.GENERAL.MANUAL_SELECTED )
      I_Contact( "DB2001_MODES_GENERAL".MG1.GENERAL.OPTIONS.SGM )
      wire#w3
      Coil( #SP.HMI_JOG_PLUS_CMM )
   END_RUNG
   RUNG wire#powerrail
      Contact( #SP.SPEED_REACHED )
      Contact( "M_DUMMY_OFF" )
   END_RUNG wire#w1
   RUNG wire#w2
      Contact( "DB2001_MODES_GENERAL".MG1.GENERAL.JOG_SELECTED )
      Contact( "DB2001_MODES_GENERAL".MG1.GENERAL.OPTIONS.SGM )
   END_RUNG wire#w3
   RUNG wire#w3
      I_Contact( #OPTIMIZATION_BYPASS )
      I_Contact( #DESELECT_SPINDLE_STO )
      { S7_Templates := "time_type := Time" } #TIMER_COMMAND_JOG_PLUS.TON(pt := #TIMER_COMMAND_JOG_PLUS.PT, et =>)
      Coil( #SpindleDB.A_Plus )
   END_RUNG
   // the same network as SCL:
   #SP.HMI_JOG_PLUS_CMM := (#SP.HMI_JOG_PLUS_RQ OR (#SP.SPEED_REACHED AND "M_DUMMY_OFF")) AND "LBP_ModeGroup".E_JOG AND NOT #SP.HMI_JOG_MINUS_CMM AND (("DB2001_MODES_GENERAL".MG1.GENERAL.MANUAL_SELECTED AND NOT "DB2001_MODES_GENERAL".MG1.GENERAL.OPTIONS.SGM) OR ("DB2001_MODES_GENERAL".MG1.GENERAL.JOG_SELECTED AND "DB2001_MODES_GENERAL".MG1.GENERAL.OPTIONS.SGM));
   #TIMER_COMMAND_JOG_PLUS(IN := #SP.HMI_JOG_PLUS_CMM AND NOT #OPTIMIZATION_BYPASS AND NOT #DESELECT_SPINDLE_STO,   // TON
                           PT := #TIMER_COMMAND_JOG_PLUS.PT);
   #SpindleDB.A_Plus := #TIMER_COMMAND_JOG_PLUS.Q;
END_REGION

REGION Network 20: OVERRIDE / FEED OVERRIDE
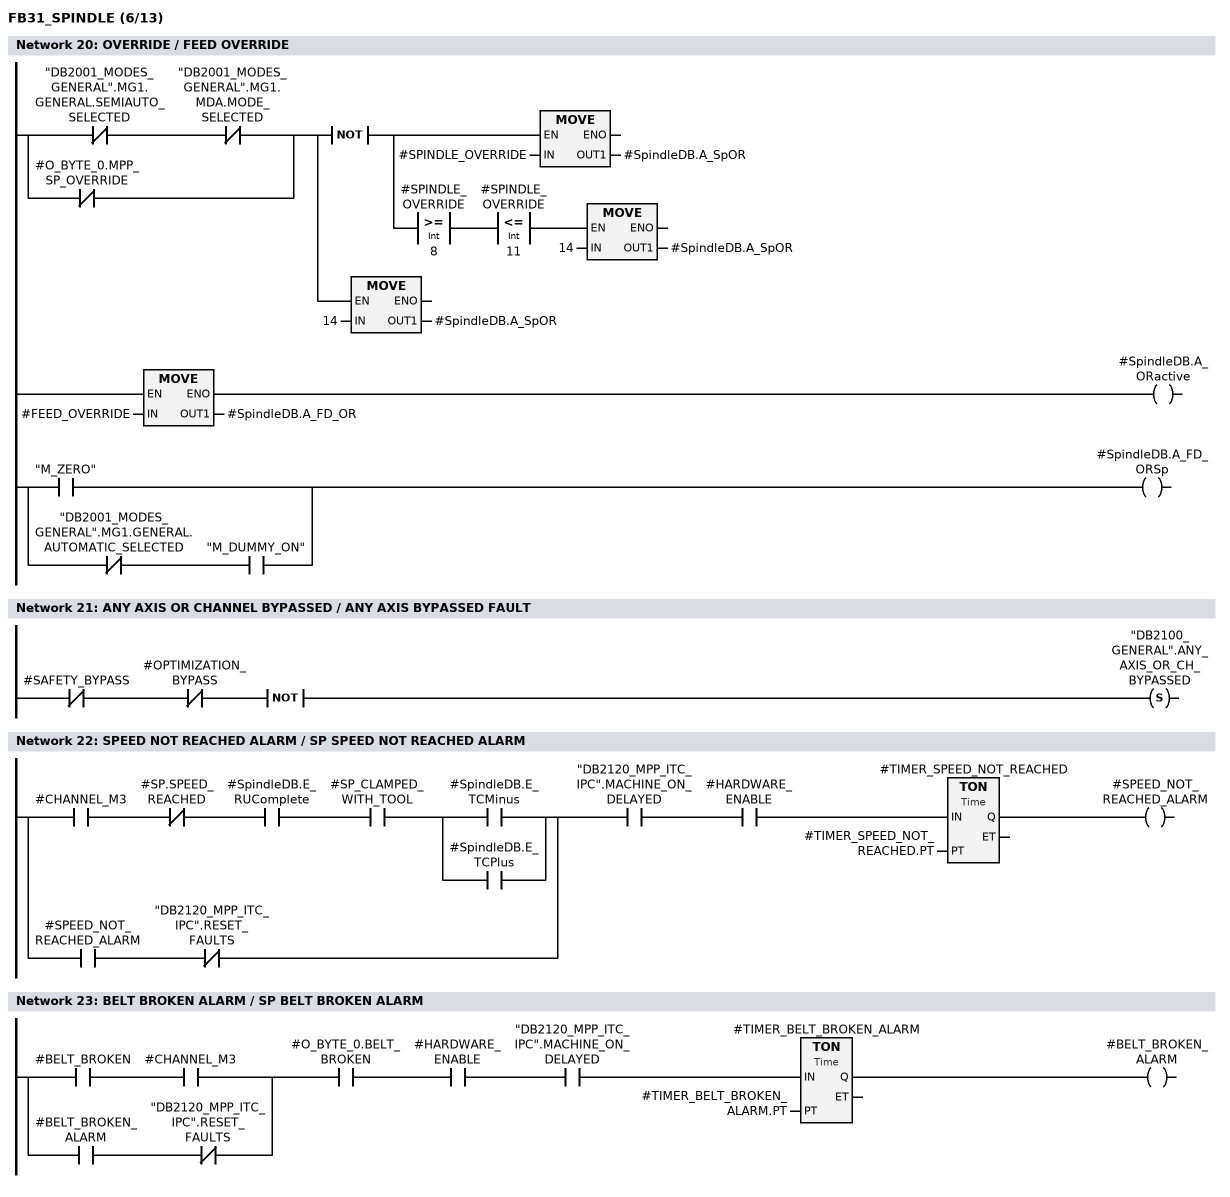
   RUNG wire#powerrail
      I_Contact( "DB2001_MODES_GENERAL".MG1.GENERAL.SEMIAUTO_SELECTED )
      I_Contact( "DB2001_MODES_GENERAL".MG1.MDA.MODE_SELECTED )
      wire#w1
      Not()
      wire#w2
      { S7_GenerateENO := "TRUE" } Move(in := #SPINDLE_OVERRIDE, out1 => #SpindleDB.A_SpOR)
   END_RUNG
   RUNG wire#powerrail
      I_Contact( #O_BYTE_0.MPP_SP_OVERRIDE )
   END_RUNG wire#w1
   RUNG wire#w2
      { S7_Templates := "SrcType := Int" } GE_Contact(in1 := #SPINDLE_OVERRIDE, in2 := 8)
      { S7_Templates := "SrcType := Int" } LE_Contact(in1 := #SPINDLE_OVERRIDE, in2 := 11)
      { S7_GenerateENO := "TRUE" } Move(in := 14, out1 => #SpindleDB.A_SpOR)
   END_RUNG
   RUNG wire#w1
      { S7_GenerateENO := "TRUE" } Move(in := 14, out1 => #SpindleDB.A_SpOR)
   END_RUNG
   RUNG wire#powerrail
      { S7_GenerateENO := "TRUE" } Move(in := #FEED_OVERRIDE, out1 => #SpindleDB.A_FD_OR)
      Coil( #SpindleDB.A_ORactive )
   END_RUNG
   RUNG wire#powerrail
      Contact( "M_ZERO" )
      wire#w3
      Coil( #SpindleDB.A_FD_ORSp )
   END_RUNG
   RUNG wire#powerrail
      I_Contact( "DB2001_MODES_GENERAL".MG1.GENERAL.AUTOMATIC_SELECTED )
      Contact( "M_DUMMY_ON" )
   END_RUNG wire#w3
   // the same network as SCL:
   // ENO of a box is taken as its EN; it also drops when the box reports an error
   #_w1 := (NOT "DB2001_MODES_GENERAL".MG1.GENERAL.SEMIAUTO_SELECTED AND NOT "DB2001_MODES_GENERAL".MG1.MDA.MODE_SELECTED) OR NOT #O_BYTE_0.MPP_SP_OVERRIDE;
   IF NOT #_w1 THEN #SpindleDB.A_SpOR := #SPINDLE_OVERRIDE; END_IF;
   IF NOT #_w1 AND (#SPINDLE_OVERRIDE >= 8) AND (#SPINDLE_OVERRIDE <= 11) THEN
       #SpindleDB.A_SpOR := 14;
   END_IF;
   IF #_w1 THEN #SpindleDB.A_SpOR := 14; END_IF;
   #SpindleDB.A_FD_OR := #FEED_OVERRIDE;
   #SpindleDB.A_ORactive := TRUE;
   #SpindleDB.A_FD_ORSp := "M_ZERO" OR (NOT "DB2001_MODES_GENERAL".MG1.GENERAL.AUTOMATIC_SELECTED AND "M_DUMMY_ON");
END_REGION

REGION Network 21: ANY AXIS OR CHANNEL BYPASSED / ANY AXIS BYPASSED FAULT
   RUNG wire#powerrail
      I_Contact( #SAFETY_BYPASS )
      I_Contact( #OPTIMIZATION_BYPASS )
      Not()
      S_Coil( "DB2100_GENERAL".ANY_AXIS_OR_CH_BYPASSED )
   END_RUNG
   // the same network as SCL:
   IF NOT (NOT #SAFETY_BYPASS AND NOT #OPTIMIZATION_BYPASS) THEN
       "DB2100_GENERAL".ANY_AXIS_OR_CH_BYPASSED := TRUE;
   END_IF;
END_REGION

REGION Network 22: SPEED NOT REACHED ALARM / SP SPEED NOT REACHED ALARM
   RUNG wire#powerrail
      Contact( #CHANNEL_M3 )
      I_Contact( #SP.SPEED_REACHED )
      Contact( #SpindleDB.E_RUComplete )
      Contact( #SP_CLAMPED_WITH_TOOL )
      wire#w1
      Contact( #SpindleDB.E_TCMinus )
      wire#w2
      Contact( "DB2120_MPP_ITC_IPC".MACHINE_ON_DELAYED )
      Contact( #HARDWARE_ENABLE )
      { S7_Templates := "time_type := Time" } #TIMER_SPEED_NOT_REACHED.TON(pt := #TIMER_SPEED_NOT_REACHED.PT, et =>)
      Coil( #SPEED_NOT_REACHED_ALARM )
   END_RUNG
   RUNG wire#w1
      Contact( #SpindleDB.E_TCPlus )
   END_RUNG wire#w2
   RUNG wire#powerrail
      Contact( #SPEED_NOT_REACHED_ALARM )
      I_Contact( "DB2120_MPP_ITC_IPC".RESET_FAULTS )
   END_RUNG wire#w2
   // the same network as SCL:
   #TIMER_SPEED_NOT_REACHED(IN := ((#CHANNEL_M3 AND NOT #SP.SPEED_REACHED AND #SpindleDB.E_RUComplete AND #SP_CLAMPED_WITH_TOOL AND (#SpindleDB.E_TCMinus OR #SpindleDB.E_TCPlus)) OR (#SPEED_NOT_REACHED_ALARM AND NOT "DB2120_MPP_ITC_IPC".RESET_FAULTS)) AND "DB2120_MPP_ITC_IPC".MACHINE_ON_DELAYED AND #HARDWARE_ENABLE,   // TON
                           PT := #TIMER_SPEED_NOT_REACHED.PT);
   #SPEED_NOT_REACHED_ALARM := #TIMER_SPEED_NOT_REACHED.Q;
END_REGION

REGION Network 23: BELT BROKEN ALARM / SP BELT BROKEN ALARM
   RUNG wire#powerrail
      Contact( #BELT_BROKEN )
      Contact( #CHANNEL_M3 )
      wire#w1
      Contact( #O_BYTE_0.BELT_BROKEN )
      Contact( #HARDWARE_ENABLE )
      Contact( "DB2120_MPP_ITC_IPC".MACHINE_ON_DELAYED )
      { S7_Templates := "time_type := Time" } #TIMER_BELT_BROKEN_ALARM.TON(pt := #TIMER_BELT_BROKEN_ALARM.PT, et =>)
      Coil( #BELT_BROKEN_ALARM )
   END_RUNG
   RUNG wire#powerrail
      Contact( #BELT_BROKEN_ALARM )
      I_Contact( "DB2120_MPP_ITC_IPC".RESET_FAULTS )
   END_RUNG wire#w1
   // the same network as SCL:
   #TIMER_BELT_BROKEN_ALARM(IN := ((#BELT_BROKEN AND #CHANNEL_M3) OR (#BELT_BROKEN_ALARM AND NOT "DB2120_MPP_ITC_IPC".RESET_FAULTS)) AND #O_BYTE_0.BELT_BROKEN AND #HARDWARE_ENABLE AND "DB2120_MPP_ITC_IPC".MACHINE_ON_DELAYED,   // TON
                           PT := #TIMER_BELT_BROKEN_ALARM.PT);
   #BELT_BROKEN_ALARM := #TIMER_BELT_BROKEN_ALARM.Q;
END_REGION

REGION Network 24: COOLING ALARM / SP COOLING ALARM
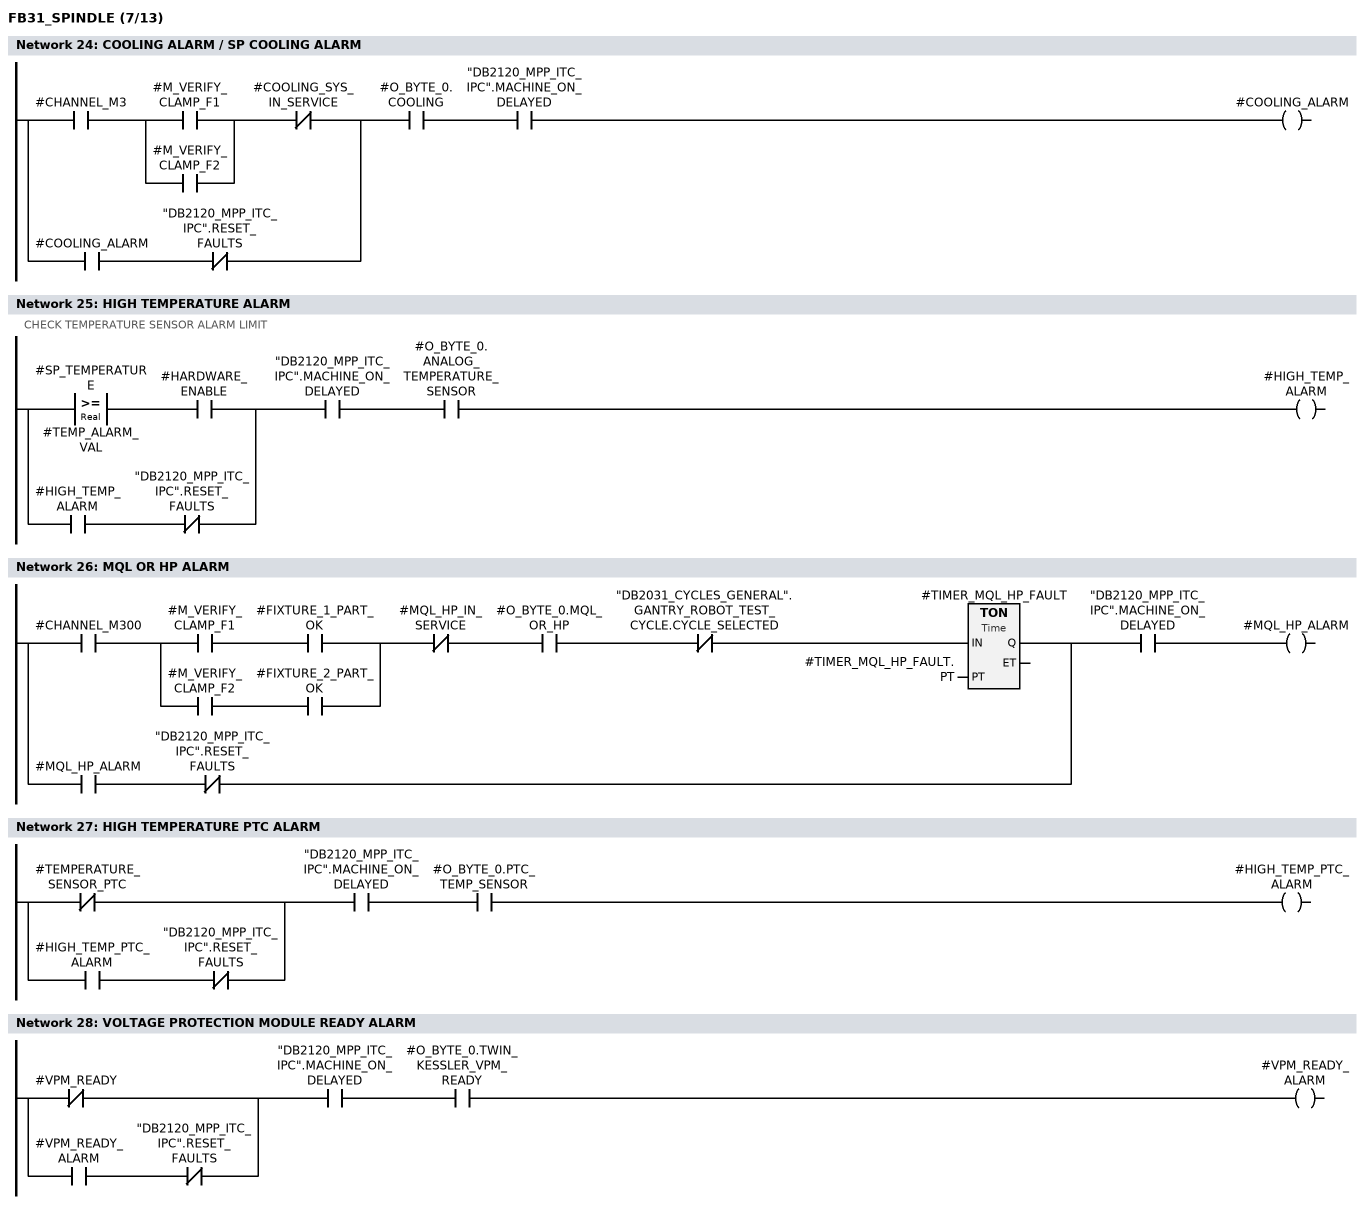
   RUNG wire#powerrail
      Contact( #CHANNEL_M3 )
      wire#w1
      Contact( #M_VERIFY_CLAMP_F1 )
      wire#w2
      I_Contact( #COOLING_SYS_IN_SERVICE )
      wire#w3
      Contact( #O_BYTE_0.COOLING )
      Contact( "DB2120_MPP_ITC_IPC".MACHINE_ON_DELAYED )
      Coil( #COOLING_ALARM )
   END_RUNG
   RUNG wire#w1
      Contact( #M_VERIFY_CLAMP_F2 )
   END_RUNG wire#w2
   RUNG wire#powerrail
      Contact( #COOLING_ALARM )
      I_Contact( "DB2120_MPP_ITC_IPC".RESET_FAULTS )
   END_RUNG wire#w3
   // the same network as SCL:
   #COOLING_ALARM := ((#CHANNEL_M3 AND (#M_VERIFY_CLAMP_F1 OR #M_VERIFY_CLAMP_F2) AND NOT #COOLING_SYS_IN_SERVICE) OR (#COOLING_ALARM AND NOT "DB2120_MPP_ITC_IPC".RESET_FAULTS)) AND #O_BYTE_0.COOLING AND "DB2120_MPP_ITC_IPC".MACHINE_ON_DELAYED;
END_REGION

REGION Network 25: HIGH TEMPERATURE ALARM
   // CHECK TEMPERATURE SENSOR ALARM LIMIT
   RUNG wire#powerrail
      { S7_Templates := "SrcType := Real" } GE_Contact(in1 := #SP_TEMPERATURE, in2 := #TEMP_ALARM_VAL)
      Contact( #HARDWARE_ENABLE )
      wire#w1
      Contact( "DB2120_MPP_ITC_IPC".MACHINE_ON_DELAYED )
      Contact( #O_BYTE_0.ANALOG_TEMPERATURE_SENSOR )
      Coil( #HIGH_TEMP_ALARM )
   END_RUNG
   RUNG wire#powerrail
      Contact( #HIGH_TEMP_ALARM )
      I_Contact( "DB2120_MPP_ITC_IPC".RESET_FAULTS )
   END_RUNG wire#w1
   // the same network as SCL:
   #HIGH_TEMP_ALARM := (((#SP_TEMPERATURE >= #TEMP_ALARM_VAL) AND #HARDWARE_ENABLE) OR (#HIGH_TEMP_ALARM AND NOT "DB2120_MPP_ITC_IPC".RESET_FAULTS)) AND "DB2120_MPP_ITC_IPC".MACHINE_ON_DELAYED AND #O_BYTE_0.ANALOG_TEMPERATURE_SENSOR;
END_REGION

REGION Network 26: MQL OR HP ALARM
   RUNG wire#powerrail
      Contact( #CHANNEL_M300 )
      wire#w1
      Contact( #M_VERIFY_CLAMP_F1 )
      Contact( #FIXTURE_1_PART_OK )
      wire#w2
      I_Contact( #MQL_HP_IN_SERVICE )
      Contact( #O_BYTE_0.MQL_OR_HP )
      I_Contact( "DB2031_CYCLES_GENERAL".GANTRY_ROBOT_TEST_CYCLE.CYCLE_SELECTED )
      { S7_Templates := "time_type := Time" } #TIMER_MQL_HP_FAULT.TON(pt := #TIMER_MQL_HP_FAULT.PT, et =>)
      wire#w3
      Contact( "DB2120_MPP_ITC_IPC".MACHINE_ON_DELAYED )
      Coil( #MQL_HP_ALARM )
   END_RUNG
   RUNG wire#w1
      Contact( #M_VERIFY_CLAMP_F2 )
      Contact( #FIXTURE_2_PART_OK )
   END_RUNG wire#w2
   RUNG wire#powerrail
      Contact( #MQL_HP_ALARM )
      I_Contact( "DB2120_MPP_ITC_IPC".RESET_FAULTS )
   END_RUNG wire#w3
   // the same network as SCL:
   #TIMER_MQL_HP_FAULT(IN := #CHANNEL_M300 AND ((#M_VERIFY_CLAMP_F1 AND #FIXTURE_1_PART_OK) OR (#M_VERIFY_CLAMP_F2 AND #FIXTURE_2_PART_OK)) AND NOT #MQL_HP_IN_SERVICE AND #O_BYTE_0.MQL_OR_HP AND NOT "DB2031_CYCLES_GENERAL".GANTRY_ROBOT_TEST_CYCLE.CYCLE_SELECTED,   // TON
                       PT := #TIMER_MQL_HP_FAULT.PT);
   #MQL_HP_ALARM := (#TIMER_MQL_HP_FAULT.Q OR (#MQL_HP_ALARM AND NOT "DB2120_MPP_ITC_IPC".RESET_FAULTS)) AND "DB2120_MPP_ITC_IPC".MACHINE_ON_DELAYED;
END_REGION

REGION Network 27: HIGH TEMPERATURE PTC ALARM
   RUNG wire#powerrail
      I_Contact( #TEMPERATURE_SENSOR_PTC )
      wire#w1
      Contact( "DB2120_MPP_ITC_IPC".MACHINE_ON_DELAYED )
      Contact( #O_BYTE_0.PTC_TEMP_SENSOR )
      Coil( #HIGH_TEMP_PTC_ALARM )
   END_RUNG
   RUNG wire#powerrail
      Contact( #HIGH_TEMP_PTC_ALARM )
      I_Contact( "DB2120_MPP_ITC_IPC".RESET_FAULTS )
   END_RUNG wire#w1
   // the same network as SCL:
   #HIGH_TEMP_PTC_ALARM := (NOT #TEMPERATURE_SENSOR_PTC OR (#HIGH_TEMP_PTC_ALARM AND NOT "DB2120_MPP_ITC_IPC".RESET_FAULTS)) AND "DB2120_MPP_ITC_IPC".MACHINE_ON_DELAYED AND #O_BYTE_0.PTC_TEMP_SENSOR;
END_REGION

REGION Network 28: VOLTAGE PROTECTION MODULE READY ALARM
   RUNG wire#powerrail
      I_Contact( #VPM_READY )
      wire#w1
      Contact( "DB2120_MPP_ITC_IPC".MACHINE_ON_DELAYED )
      Contact( #O_BYTE_0.TWIN_KESSLER_VPM_READY )
      Coil( #VPM_READY_ALARM )
   END_RUNG
   RUNG wire#powerrail
      Contact( #VPM_READY_ALARM )
      I_Contact( "DB2120_MPP_ITC_IPC".RESET_FAULTS )
   END_RUNG wire#w1
   // the same network as SCL:
   #VPM_READY_ALARM := (NOT #VPM_READY OR (#VPM_READY_ALARM AND NOT "DB2120_MPP_ITC_IPC".RESET_FAULTS)) AND "DB2120_MPP_ITC_IPC".MACHINE_ON_DELAYED AND #O_BYTE_0.TWIN_KESSLER_VPM_READY;
END_REGION

REGION Network 29: RETURN HOME POSITION AND STOP END OF CYCLE ALARMS / RHP&SEOC ALARMS
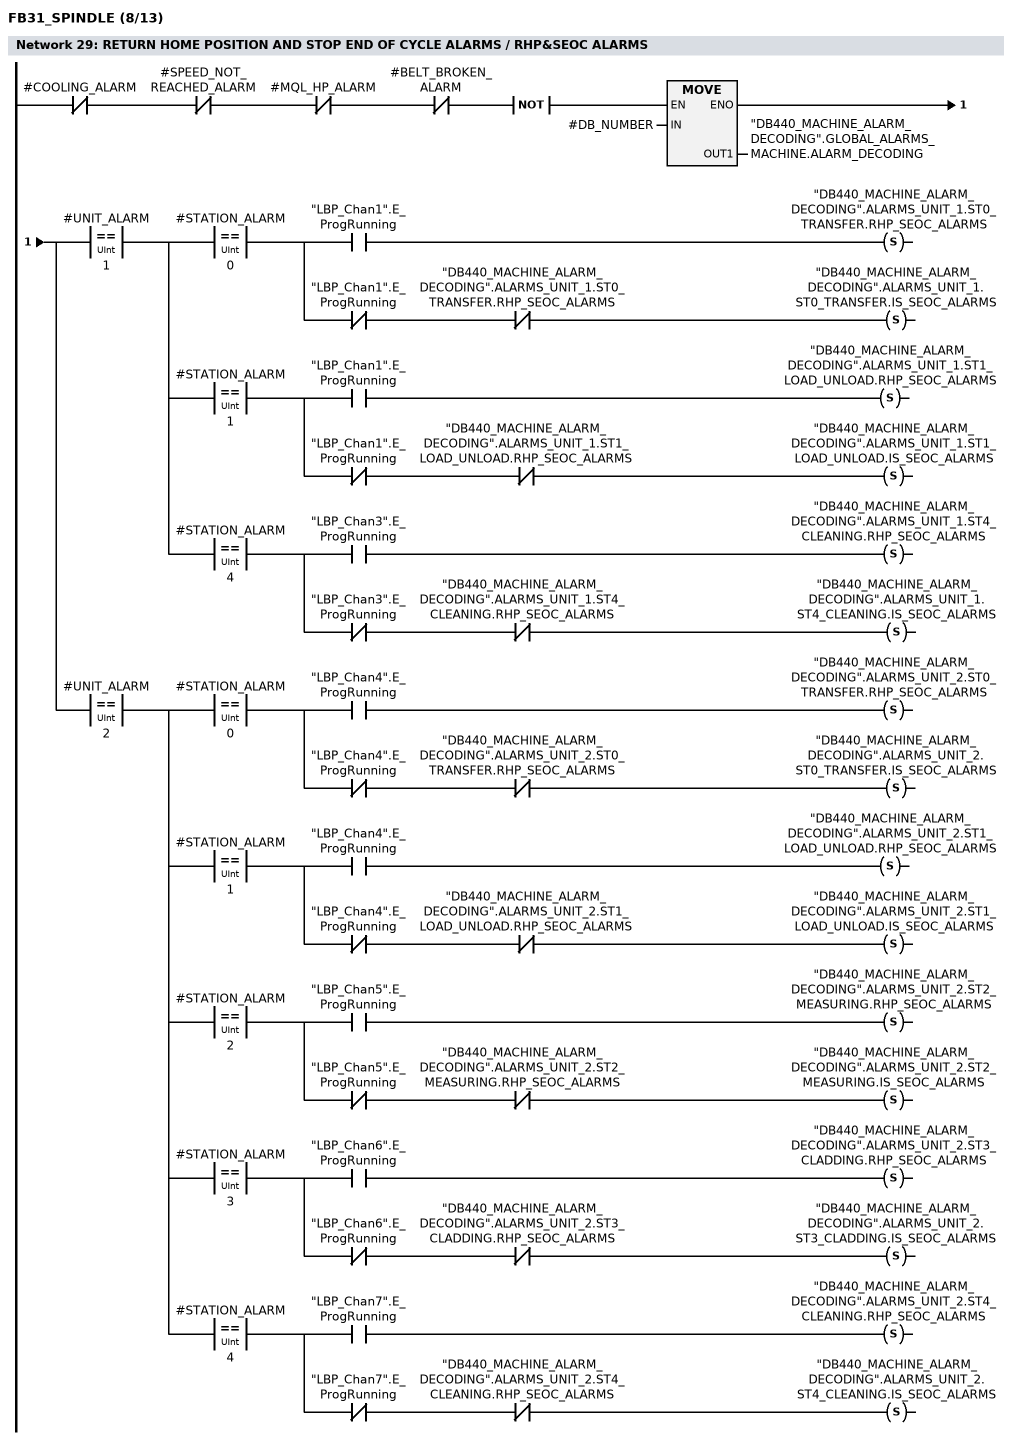
   RUNG wire#powerrail
      I_Contact( #COOLING_ALARM )
      I_Contact( #SPEED_NOT_REACHED_ALARM )
      I_Contact( #MQL_HP_ALARM )
      I_Contact( #BELT_BROKEN_ALARM )
      Not()
      { S7_GenerateENO := "TRUE" } Move(in := #DB_NUMBER, out1 => "DB440_MACHINE_ALARM_DECODING".GLOBAL_ALARMS_MACHINE.ALARM_DECODING)
      wire#w1
      { S7_Templates := "SrcType := UInt" } EQ_Contact(in1 := #UNIT_ALARM, in2 := 1)
      wire#w2
      { S7_Templates := "SrcType := UInt" } EQ_Contact(in1 := #STATION_ALARM, in2 := 0)
      wire#w3
      Contact( "LBP_Chan1".E_ProgRunning )
      S_Coil( "DB440_MACHINE_ALARM_DECODING".ALARMS_UNIT_1.ST0_TRANSFER.RHP_SEOC_ALARMS )
   END_RUNG
   RUNG wire#w3
      I_Contact( "LBP_Chan1".E_ProgRunning )
      I_Contact( "DB440_MACHINE_ALARM_DECODING".ALARMS_UNIT_1.ST0_TRANSFER.RHP_SEOC_ALARMS )
      S_Coil( "DB440_MACHINE_ALARM_DECODING".ALARMS_UNIT_1.ST0_TRANSFER.IS_SEOC_ALARMS )
   END_RUNG
   RUNG wire#w2
      { S7_Templates := "SrcType := UInt" } EQ_Contact(in1 := #STATION_ALARM, in2 := 1)
      wire#w4
      Contact( "LBP_Chan1".E_ProgRunning )
      S_Coil( "DB440_MACHINE_ALARM_DECODING".ALARMS_UNIT_1.ST1_LOAD_UNLOAD.RHP_SEOC_ALARMS )
   END_RUNG
   RUNG wire#w4
      I_Contact( "LBP_Chan1".E_ProgRunning )
      I_Contact( "DB440_MACHINE_ALARM_DECODING".ALARMS_UNIT_1.ST1_LOAD_UNLOAD.RHP_SEOC_ALARMS )
      S_Coil( "DB440_MACHINE_ALARM_DECODING".ALARMS_UNIT_1.ST1_LOAD_UNLOAD.IS_SEOC_ALARMS )
   END_RUNG
   RUNG wire#w2
      { S7_Templates := "SrcType := UInt" } EQ_Contact(in1 := #STATION_ALARM, in2 := 4)
      wire#w5
      Contact( "LBP_Chan3".E_ProgRunning )
      S_Coil( "DB440_MACHINE_ALARM_DECODING".ALARMS_UNIT_1.ST4_CLEANING.RHP_SEOC_ALARMS )
   END_RUNG
   RUNG wire#w5
      I_Contact( "LBP_Chan3".E_ProgRunning )
      I_Contact( "DB440_MACHINE_ALARM_DECODING".ALARMS_UNIT_1.ST4_CLEANING.RHP_SEOC_ALARMS )
      S_Coil( "DB440_MACHINE_ALARM_DECODING".ALARMS_UNIT_1.ST4_CLEANING.IS_SEOC_ALARMS )
   END_RUNG
   RUNG wire#w1
      { S7_Templates := "SrcType := UInt" } EQ_Contact(in1 := #UNIT_ALARM, in2 := 2)
      wire#w6
      { S7_Templates := "SrcType := UInt" } EQ_Contact(in1 := #STATION_ALARM, in2 := 0)
      wire#w7
      Contact( "LBP_Chan4".E_ProgRunning )
      S_Coil( "DB440_MACHINE_ALARM_DECODING".ALARMS_UNIT_2.ST0_TRANSFER.RHP_SEOC_ALARMS )
   END_RUNG
   RUNG wire#w7
      I_Contact( "LBP_Chan4".E_ProgRunning )
      I_Contact( "DB440_MACHINE_ALARM_DECODING".ALARMS_UNIT_2.ST0_TRANSFER.RHP_SEOC_ALARMS )
      S_Coil( "DB440_MACHINE_ALARM_DECODING".ALARMS_UNIT_2.ST0_TRANSFER.IS_SEOC_ALARMS )
   END_RUNG
   RUNG wire#w6
      { S7_Templates := "SrcType := UInt" } EQ_Contact(in1 := #STATION_ALARM, in2 := 1)
      wire#w8
      Contact( "LBP_Chan4".E_ProgRunning )
      S_Coil( "DB440_MACHINE_ALARM_DECODING".ALARMS_UNIT_2.ST1_LOAD_UNLOAD.RHP_SEOC_ALARMS )
   END_RUNG
   RUNG wire#w8
      I_Contact( "LBP_Chan4".E_ProgRunning )
      I_Contact( "DB440_MACHINE_ALARM_DECODING".ALARMS_UNIT_2.ST1_LOAD_UNLOAD.RHP_SEOC_ALARMS )
      S_Coil( "DB440_MACHINE_ALARM_DECODING".ALARMS_UNIT_2.ST1_LOAD_UNLOAD.IS_SEOC_ALARMS )
   END_RUNG
   RUNG wire#w6
      { S7_Templates := "SrcType := UInt" } EQ_Contact(in1 := #STATION_ALARM, in2 := 2)
      wire#w9
      Contact( "LBP_Chan5".E_ProgRunning )
      S_Coil( "DB440_MACHINE_ALARM_DECODING".ALARMS_UNIT_2.ST2_MEASURING.RHP_SEOC_ALARMS )
   END_RUNG
   RUNG wire#w9
      I_Contact( "LBP_Chan5".E_ProgRunning )
      I_Contact( "DB440_MACHINE_ALARM_DECODING".ALARMS_UNIT_2.ST2_MEASURING.RHP_SEOC_ALARMS )
      S_Coil( "DB440_MACHINE_ALARM_DECODING".ALARMS_UNIT_2.ST2_MEASURING.IS_SEOC_ALARMS )
   END_RUNG
   RUNG wire#w6
      { S7_Templates := "SrcType := UInt" } EQ_Contact(in1 := #STATION_ALARM, in2 := 3)
      wire#w10
      Contact( "LBP_Chan6".E_ProgRunning )
      S_Coil( "DB440_MACHINE_ALARM_DECODING".ALARMS_UNIT_2.ST3_CLADDING.RHP_SEOC_ALARMS )
   END_RUNG
   RUNG wire#w10
      I_Contact( "LBP_Chan6".E_ProgRunning )
      I_Contact( "DB440_MACHINE_ALARM_DECODING".ALARMS_UNIT_2.ST3_CLADDING.RHP_SEOC_ALARMS )
      S_Coil( "DB440_MACHINE_ALARM_DECODING".ALARMS_UNIT_2.ST3_CLADDING.IS_SEOC_ALARMS )
   END_RUNG
   RUNG wire#w6
      { S7_Templates := "SrcType := UInt" } EQ_Contact(in1 := #STATION_ALARM, in2 := 4)
      wire#w11
      Contact( "LBP_Chan7".E_ProgRunning )
      S_Coil( "DB440_MACHINE_ALARM_DECODING".ALARMS_UNIT_2.ST4_CLEANING.RHP_SEOC_ALARMS )
   END_RUNG
   RUNG wire#w11
      I_Contact( "LBP_Chan7".E_ProgRunning )
      I_Contact( "DB440_MACHINE_ALARM_DECODING".ALARMS_UNIT_2.ST4_CLEANING.RHP_SEOC_ALARMS )
      S_Coil( "DB440_MACHINE_ALARM_DECODING".ALARMS_UNIT_2.ST4_CLEANING.IS_SEOC_ALARMS )
   END_RUNG
   // the same network as SCL:
   // ENO of a box is taken as its EN; it also drops when the box reports an error
   #_w1 := NOT (NOT #COOLING_ALARM AND NOT #SPEED_NOT_REACHED_ALARM AND NOT #MQL_HP_ALARM AND NOT #BELT_BROKEN_ALARM);
   IF #_w1 THEN "DB440_MACHINE_ALARM_DECODING".GLOBAL_ALARMS_MACHINE.ALARM_DECODING := #DB_NUMBER; END_IF;
   #_w2 := #_w1 AND (#UNIT_ALARM = 1);
   #_w3 := #_w2 AND (#STATION_ALARM = 0);
   IF #_w3 AND "LBP_Chan1".E_ProgRunning THEN
       "DB440_MACHINE_ALARM_DECODING".ALARMS_UNIT_1.ST0_TRANSFER.RHP_SEOC_ALARMS := TRUE;
   END_IF;
   IF #_w3 AND NOT "LBP_Chan1".E_ProgRunning AND NOT "DB440_MACHINE_ALARM_DECODING".ALARMS_UNIT_1.ST0_TRANSFER.RHP_SEOC_ALARMS THEN
       "DB440_MACHINE_ALARM_DECODING".ALARMS_UNIT_1.ST0_TRANSFER.IS_SEOC_ALARMS := TRUE;
   END_IF;
   #_w4 := #_w2 AND (#STATION_ALARM = 1);
   IF #_w4 AND "LBP_Chan1".E_ProgRunning THEN
       "DB440_MACHINE_ALARM_DECODING".ALARMS_UNIT_1.ST1_LOAD_UNLOAD.RHP_SEOC_ALARMS := TRUE;
   END_IF;
   IF #_w4 AND NOT "LBP_Chan1".E_ProgRunning AND NOT "DB440_MACHINE_ALARM_DECODING".ALARMS_UNIT_1.ST1_LOAD_UNLOAD.RHP_SEOC_ALARMS THEN
       "DB440_MACHINE_ALARM_DECODING".ALARMS_UNIT_1.ST1_LOAD_UNLOAD.IS_SEOC_ALARMS := TRUE;
   END_IF;
   #_w5 := #_w2 AND (#STATION_ALARM = 4);
   IF #_w5 AND "LBP_Chan3".E_ProgRunning THEN
       "DB440_MACHINE_ALARM_DECODING".ALARMS_UNIT_1.ST4_CLEANING.RHP_SEOC_ALARMS := TRUE;
   END_IF;
   IF #_w5 AND NOT "LBP_Chan3".E_ProgRunning AND NOT "DB440_MACHINE_ALARM_DECODING".ALARMS_UNIT_1.ST4_CLEANING.RHP_SEOC_ALARMS THEN
       "DB440_MACHINE_ALARM_DECODING".ALARMS_UNIT_1.ST4_CLEANING.IS_SEOC_ALARMS := TRUE;
   END_IF;
   #_w6 := #_w1 AND (#UNIT_ALARM = 2);
   #_w7 := #_w6 AND (#STATION_ALARM = 0);
   IF #_w7 AND "LBP_Chan4".E_ProgRunning THEN
       "DB440_MACHINE_ALARM_DECODING".ALARMS_UNIT_2.ST0_TRANSFER.RHP_SEOC_ALARMS := TRUE;
   END_IF;
   IF #_w7 AND NOT "LBP_Chan4".E_ProgRunning AND NOT "DB440_MACHINE_ALARM_DECODING".ALARMS_UNIT_2.ST0_TRANSFER.RHP_SEOC_ALARMS THEN
       "DB440_MACHINE_ALARM_DECODING".ALARMS_UNIT_2.ST0_TRANSFER.IS_SEOC_ALARMS := TRUE;
   END_IF;
   #_w8 := #_w6 AND (#STATION_ALARM = 1);
   IF #_w8 AND "LBP_Chan4".E_ProgRunning THEN
       "DB440_MACHINE_ALARM_DECODING".ALARMS_UNIT_2.ST1_LOAD_UNLOAD.RHP_SEOC_ALARMS := TRUE;
   END_IF;
   IF #_w8 AND NOT "LBP_Chan4".E_ProgRunning AND NOT "DB440_MACHINE_ALARM_DECODING".ALARMS_UNIT_2.ST1_LOAD_UNLOAD.RHP_SEOC_ALARMS THEN
       "DB440_MACHINE_ALARM_DECODING".ALARMS_UNIT_2.ST1_LOAD_UNLOAD.IS_SEOC_ALARMS := TRUE;
   END_IF;
   #_w9 := #_w6 AND (#STATION_ALARM = 2);
   IF #_w9 AND "LBP_Chan5".E_ProgRunning THEN
       "DB440_MACHINE_ALARM_DECODING".ALARMS_UNIT_2.ST2_MEASURING.RHP_SEOC_ALARMS := TRUE;
   END_IF;
   IF #_w9 AND NOT "LBP_Chan5".E_ProgRunning AND NOT "DB440_MACHINE_ALARM_DECODING".ALARMS_UNIT_2.ST2_MEASURING.RHP_SEOC_ALARMS THEN
       "DB440_MACHINE_ALARM_DECODING".ALARMS_UNIT_2.ST2_MEASURING.IS_SEOC_ALARMS := TRUE;
   END_IF;
   #_w10 := #_w6 AND (#STATION_ALARM = 3);
   IF #_w10 AND "LBP_Chan6".E_ProgRunning THEN
       "DB440_MACHINE_ALARM_DECODING".ALARMS_UNIT_2.ST3_CLADDING.RHP_SEOC_ALARMS := TRUE;
   END_IF;
   IF #_w10 AND NOT "LBP_Chan6".E_ProgRunning AND NOT "DB440_MACHINE_ALARM_DECODING".ALARMS_UNIT_2.ST3_CLADDING.RHP_SEOC_ALARMS THEN
       "DB440_MACHINE_ALARM_DECODING".ALARMS_UNIT_2.ST3_CLADDING.IS_SEOC_ALARMS := TRUE;
   END_IF;
   #_w11 := #_w6 AND (#STATION_ALARM = 4);
   IF #_w11 AND "LBP_Chan7".E_ProgRunning THEN
       "DB440_MACHINE_ALARM_DECODING".ALARMS_UNIT_2.ST4_CLEANING.RHP_SEOC_ALARMS := TRUE;
   END_IF;
   IF #_w11 AND NOT "LBP_Chan7".E_ProgRunning AND NOT "DB440_MACHINE_ALARM_DECODING".ALARMS_UNIT_2.ST4_CLEANING.RHP_SEOC_ALARMS THEN
       "DB440_MACHINE_ALARM_DECODING".ALARMS_UNIT_2.ST4_CLEANING.IS_SEOC_ALARMS := TRUE;
   END_IF;
END_REGION

REGION Network 30: STOP END OF CYCLE ALARMS / SEOC ALARMS
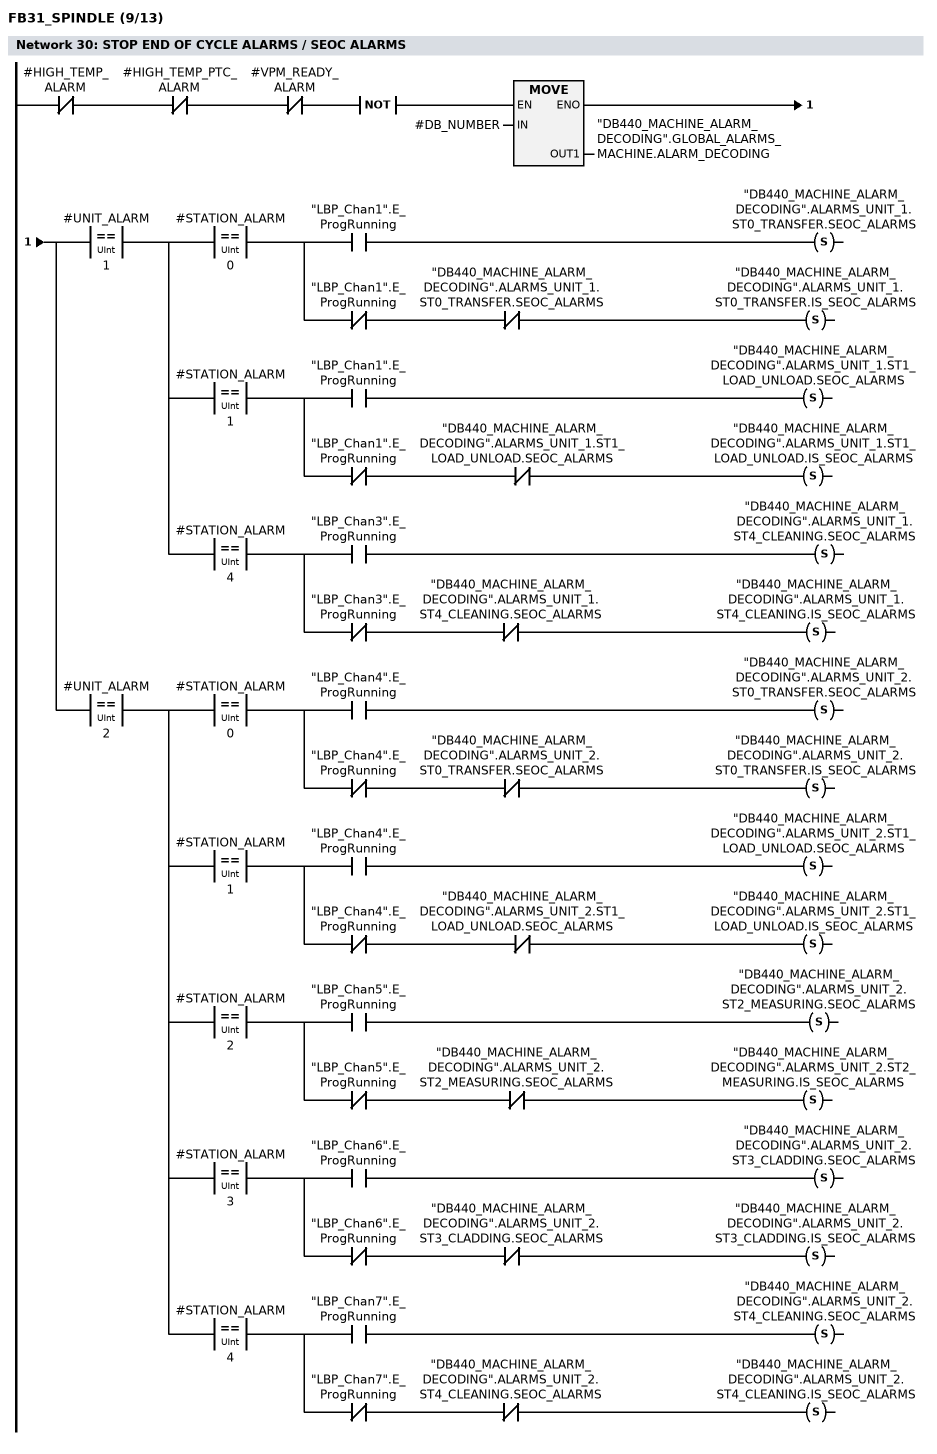
   RUNG wire#powerrail
      I_Contact( #HIGH_TEMP_ALARM )
      I_Contact( #HIGH_TEMP_PTC_ALARM )
      I_Contact( #VPM_READY_ALARM )
      Not()
      { S7_GenerateENO := "TRUE" } Move(in := #DB_NUMBER, out1 => "DB440_MACHINE_ALARM_DECODING".GLOBAL_ALARMS_MACHINE.ALARM_DECODING)
      wire#w1
      { S7_Templates := "SrcType := UInt" } EQ_Contact(in1 := #UNIT_ALARM, in2 := 1)
      wire#w2
      { S7_Templates := "SrcType := UInt" } EQ_Contact(in1 := #STATION_ALARM, in2 := 0)
      wire#w3
      Contact( "LBP_Chan1".E_ProgRunning )
      S_Coil( "DB440_MACHINE_ALARM_DECODING".ALARMS_UNIT_1.ST0_TRANSFER.SEOC_ALARMS )
   END_RUNG
   RUNG wire#w3
      I_Contact( "LBP_Chan1".E_ProgRunning )
      I_Contact( "DB440_MACHINE_ALARM_DECODING".ALARMS_UNIT_1.ST0_TRANSFER.SEOC_ALARMS )
      S_Coil( "DB440_MACHINE_ALARM_DECODING".ALARMS_UNIT_1.ST0_TRANSFER.IS_SEOC_ALARMS )
   END_RUNG
   RUNG wire#w2
      { S7_Templates := "SrcType := UInt" } EQ_Contact(in1 := #STATION_ALARM, in2 := 1)
      wire#w4
      Contact( "LBP_Chan1".E_ProgRunning )
      S_Coil( "DB440_MACHINE_ALARM_DECODING".ALARMS_UNIT_1.ST1_LOAD_UNLOAD.SEOC_ALARMS )
   END_RUNG
   RUNG wire#w4
      I_Contact( "LBP_Chan1".E_ProgRunning )
      I_Contact( "DB440_MACHINE_ALARM_DECODING".ALARMS_UNIT_1.ST1_LOAD_UNLOAD.SEOC_ALARMS )
      S_Coil( "DB440_MACHINE_ALARM_DECODING".ALARMS_UNIT_1.ST1_LOAD_UNLOAD.IS_SEOC_ALARMS )
   END_RUNG
   RUNG wire#w2
      { S7_Templates := "SrcType := UInt" } EQ_Contact(in1 := #STATION_ALARM, in2 := 4)
      wire#w5
      Contact( "LBP_Chan3".E_ProgRunning )
      S_Coil( "DB440_MACHINE_ALARM_DECODING".ALARMS_UNIT_1.ST4_CLEANING.SEOC_ALARMS )
   END_RUNG
   RUNG wire#w5
      I_Contact( "LBP_Chan3".E_ProgRunning )
      I_Contact( "DB440_MACHINE_ALARM_DECODING".ALARMS_UNIT_1.ST4_CLEANING.SEOC_ALARMS )
      S_Coil( "DB440_MACHINE_ALARM_DECODING".ALARMS_UNIT_1.ST4_CLEANING.IS_SEOC_ALARMS )
   END_RUNG
   RUNG wire#w1
      { S7_Templates := "SrcType := UInt" } EQ_Contact(in1 := #UNIT_ALARM, in2 := 2)
      wire#w6
      { S7_Templates := "SrcType := UInt" } EQ_Contact(in1 := #STATION_ALARM, in2 := 0)
      wire#w7
      Contact( "LBP_Chan4".E_ProgRunning )
      S_Coil( "DB440_MACHINE_ALARM_DECODING".ALARMS_UNIT_2.ST0_TRANSFER.SEOC_ALARMS )
   END_RUNG
   RUNG wire#w7
      I_Contact( "LBP_Chan4".E_ProgRunning )
      I_Contact( "DB440_MACHINE_ALARM_DECODING".ALARMS_UNIT_2.ST0_TRANSFER.SEOC_ALARMS )
      S_Coil( "DB440_MACHINE_ALARM_DECODING".ALARMS_UNIT_2.ST0_TRANSFER.IS_SEOC_ALARMS )
   END_RUNG
   RUNG wire#w6
      { S7_Templates := "SrcType := UInt" } EQ_Contact(in1 := #STATION_ALARM, in2 := 1)
      wire#w8
      Contact( "LBP_Chan4".E_ProgRunning )
      S_Coil( "DB440_MACHINE_ALARM_DECODING".ALARMS_UNIT_2.ST1_LOAD_UNLOAD.SEOC_ALARMS )
   END_RUNG
   RUNG wire#w8
      I_Contact( "LBP_Chan4".E_ProgRunning )
      I_Contact( "DB440_MACHINE_ALARM_DECODING".ALARMS_UNIT_2.ST1_LOAD_UNLOAD.SEOC_ALARMS )
      S_Coil( "DB440_MACHINE_ALARM_DECODING".ALARMS_UNIT_2.ST1_LOAD_UNLOAD.IS_SEOC_ALARMS )
   END_RUNG
   RUNG wire#w6
      { S7_Templates := "SrcType := UInt" } EQ_Contact(in1 := #STATION_ALARM, in2 := 2)
      wire#w9
      Contact( "LBP_Chan5".E_ProgRunning )
      S_Coil( "DB440_MACHINE_ALARM_DECODING".ALARMS_UNIT_2.ST2_MEASURING.SEOC_ALARMS )
   END_RUNG
   RUNG wire#w9
      I_Contact( "LBP_Chan5".E_ProgRunning )
      I_Contact( "DB440_MACHINE_ALARM_DECODING".ALARMS_UNIT_2.ST2_MEASURING.SEOC_ALARMS )
      S_Coil( "DB440_MACHINE_ALARM_DECODING".ALARMS_UNIT_2.ST2_MEASURING.IS_SEOC_ALARMS )
   END_RUNG
   RUNG wire#w6
      { S7_Templates := "SrcType := UInt" } EQ_Contact(in1 := #STATION_ALARM, in2 := 3)
      wire#w10
      Contact( "LBP_Chan6".E_ProgRunning )
      S_Coil( "DB440_MACHINE_ALARM_DECODING".ALARMS_UNIT_2.ST3_CLADDING.SEOC_ALARMS )
   END_RUNG
   RUNG wire#w10
      I_Contact( "LBP_Chan6".E_ProgRunning )
      I_Contact( "DB440_MACHINE_ALARM_DECODING".ALARMS_UNIT_2.ST3_CLADDING.SEOC_ALARMS )
      S_Coil( "DB440_MACHINE_ALARM_DECODING".ALARMS_UNIT_2.ST3_CLADDING.IS_SEOC_ALARMS )
   END_RUNG
   RUNG wire#w6
      { S7_Templates := "SrcType := UInt" } EQ_Contact(in1 := #STATION_ALARM, in2 := 4)
      wire#w11
      Contact( "LBP_Chan7".E_ProgRunning )
      S_Coil( "DB440_MACHINE_ALARM_DECODING".ALARMS_UNIT_2.ST4_CLEANING.SEOC_ALARMS )
   END_RUNG
   RUNG wire#w11
      I_Contact( "LBP_Chan7".E_ProgRunning )
      I_Contact( "DB440_MACHINE_ALARM_DECODING".ALARMS_UNIT_2.ST4_CLEANING.SEOC_ALARMS )
      S_Coil( "DB440_MACHINE_ALARM_DECODING".ALARMS_UNIT_2.ST4_CLEANING.IS_SEOC_ALARMS )
   END_RUNG
   // the same network as SCL:
   // ENO of a box is taken as its EN; it also drops when the box reports an error
   #_w1 := NOT (NOT #HIGH_TEMP_ALARM AND NOT #HIGH_TEMP_PTC_ALARM AND NOT #VPM_READY_ALARM);
   IF #_w1 THEN "DB440_MACHINE_ALARM_DECODING".GLOBAL_ALARMS_MACHINE.ALARM_DECODING := #DB_NUMBER; END_IF;
   #_w2 := #_w1 AND (#UNIT_ALARM = 1);
   #_w3 := #_w2 AND (#STATION_ALARM = 0);
   IF #_w3 AND "LBP_Chan1".E_ProgRunning THEN
       "DB440_MACHINE_ALARM_DECODING".ALARMS_UNIT_1.ST0_TRANSFER.SEOC_ALARMS := TRUE;
   END_IF;
   IF #_w3 AND NOT "LBP_Chan1".E_ProgRunning AND NOT "DB440_MACHINE_ALARM_DECODING".ALARMS_UNIT_1.ST0_TRANSFER.SEOC_ALARMS THEN
       "DB440_MACHINE_ALARM_DECODING".ALARMS_UNIT_1.ST0_TRANSFER.IS_SEOC_ALARMS := TRUE;
   END_IF;
   #_w4 := #_w2 AND (#STATION_ALARM = 1);
   IF #_w4 AND "LBP_Chan1".E_ProgRunning THEN
       "DB440_MACHINE_ALARM_DECODING".ALARMS_UNIT_1.ST1_LOAD_UNLOAD.SEOC_ALARMS := TRUE;
   END_IF;
   IF #_w4 AND NOT "LBP_Chan1".E_ProgRunning AND NOT "DB440_MACHINE_ALARM_DECODING".ALARMS_UNIT_1.ST1_LOAD_UNLOAD.SEOC_ALARMS THEN
       "DB440_MACHINE_ALARM_DECODING".ALARMS_UNIT_1.ST1_LOAD_UNLOAD.IS_SEOC_ALARMS := TRUE;
   END_IF;
   #_w5 := #_w2 AND (#STATION_ALARM = 4);
   IF #_w5 AND "LBP_Chan3".E_ProgRunning THEN
       "DB440_MACHINE_ALARM_DECODING".ALARMS_UNIT_1.ST4_CLEANING.SEOC_ALARMS := TRUE;
   END_IF;
   IF #_w5 AND NOT "LBP_Chan3".E_ProgRunning AND NOT "DB440_MACHINE_ALARM_DECODING".ALARMS_UNIT_1.ST4_CLEANING.SEOC_ALARMS THEN
       "DB440_MACHINE_ALARM_DECODING".ALARMS_UNIT_1.ST4_CLEANING.IS_SEOC_ALARMS := TRUE;
   END_IF;
   #_w6 := #_w1 AND (#UNIT_ALARM = 2);
   #_w7 := #_w6 AND (#STATION_ALARM = 0);
   IF #_w7 AND "LBP_Chan4".E_ProgRunning THEN
       "DB440_MACHINE_ALARM_DECODING".ALARMS_UNIT_2.ST0_TRANSFER.SEOC_ALARMS := TRUE;
   END_IF;
   IF #_w7 AND NOT "LBP_Chan4".E_ProgRunning AND NOT "DB440_MACHINE_ALARM_DECODING".ALARMS_UNIT_2.ST0_TRANSFER.SEOC_ALARMS THEN
       "DB440_MACHINE_ALARM_DECODING".ALARMS_UNIT_2.ST0_TRANSFER.IS_SEOC_ALARMS := TRUE;
   END_IF;
   #_w8 := #_w6 AND (#STATION_ALARM = 1);
   IF #_w8 AND "LBP_Chan4".E_ProgRunning THEN
       "DB440_MACHINE_ALARM_DECODING".ALARMS_UNIT_2.ST1_LOAD_UNLOAD.SEOC_ALARMS := TRUE;
   END_IF;
   IF #_w8 AND NOT "LBP_Chan4".E_ProgRunning AND NOT "DB440_MACHINE_ALARM_DECODING".ALARMS_UNIT_2.ST1_LOAD_UNLOAD.SEOC_ALARMS THEN
       "DB440_MACHINE_ALARM_DECODING".ALARMS_UNIT_2.ST1_LOAD_UNLOAD.IS_SEOC_ALARMS := TRUE;
   END_IF;
   #_w9 := #_w6 AND (#STATION_ALARM = 2);
   IF #_w9 AND "LBP_Chan5".E_ProgRunning THEN
       "DB440_MACHINE_ALARM_DECODING".ALARMS_UNIT_2.ST2_MEASURING.SEOC_ALARMS := TRUE;
   END_IF;
   IF #_w9 AND NOT "LBP_Chan5".E_ProgRunning AND NOT "DB440_MACHINE_ALARM_DECODING".ALARMS_UNIT_2.ST2_MEASURING.SEOC_ALARMS THEN
       "DB440_MACHINE_ALARM_DECODING".ALARMS_UNIT_2.ST2_MEASURING.IS_SEOC_ALARMS := TRUE;
   END_IF;
   #_w10 := #_w6 AND (#STATION_ALARM = 3);
   IF #_w10 AND "LBP_Chan6".E_ProgRunning THEN
       "DB440_MACHINE_ALARM_DECODING".ALARMS_UNIT_2.ST3_CLADDING.SEOC_ALARMS := TRUE;
   END_IF;
   IF #_w10 AND NOT "LBP_Chan6".E_ProgRunning AND NOT "DB440_MACHINE_ALARM_DECODING".ALARMS_UNIT_2.ST3_CLADDING.SEOC_ALARMS THEN
       "DB440_MACHINE_ALARM_DECODING".ALARMS_UNIT_2.ST3_CLADDING.IS_SEOC_ALARMS := TRUE;
   END_IF;
   #_w11 := #_w6 AND (#STATION_ALARM = 4);
   IF #_w11 AND "LBP_Chan7".E_ProgRunning THEN
       "DB440_MACHINE_ALARM_DECODING".ALARMS_UNIT_2.ST4_CLEANING.SEOC_ALARMS := TRUE;
   END_IF;
   IF #_w11 AND NOT "LBP_Chan7".E_ProgRunning AND NOT "DB440_MACHINE_ALARM_DECODING".ALARMS_UNIT_2.ST4_CLEANING.SEOC_ALARMS THEN
       "DB440_MACHINE_ALARM_DECODING".ALARMS_UNIT_2.ST4_CLEANING.IS_SEOC_ALARMS := TRUE;
   END_IF;
END_REGION

REGION Network 31: RETURN HOME POSITION AND RUN OUT ALARMS
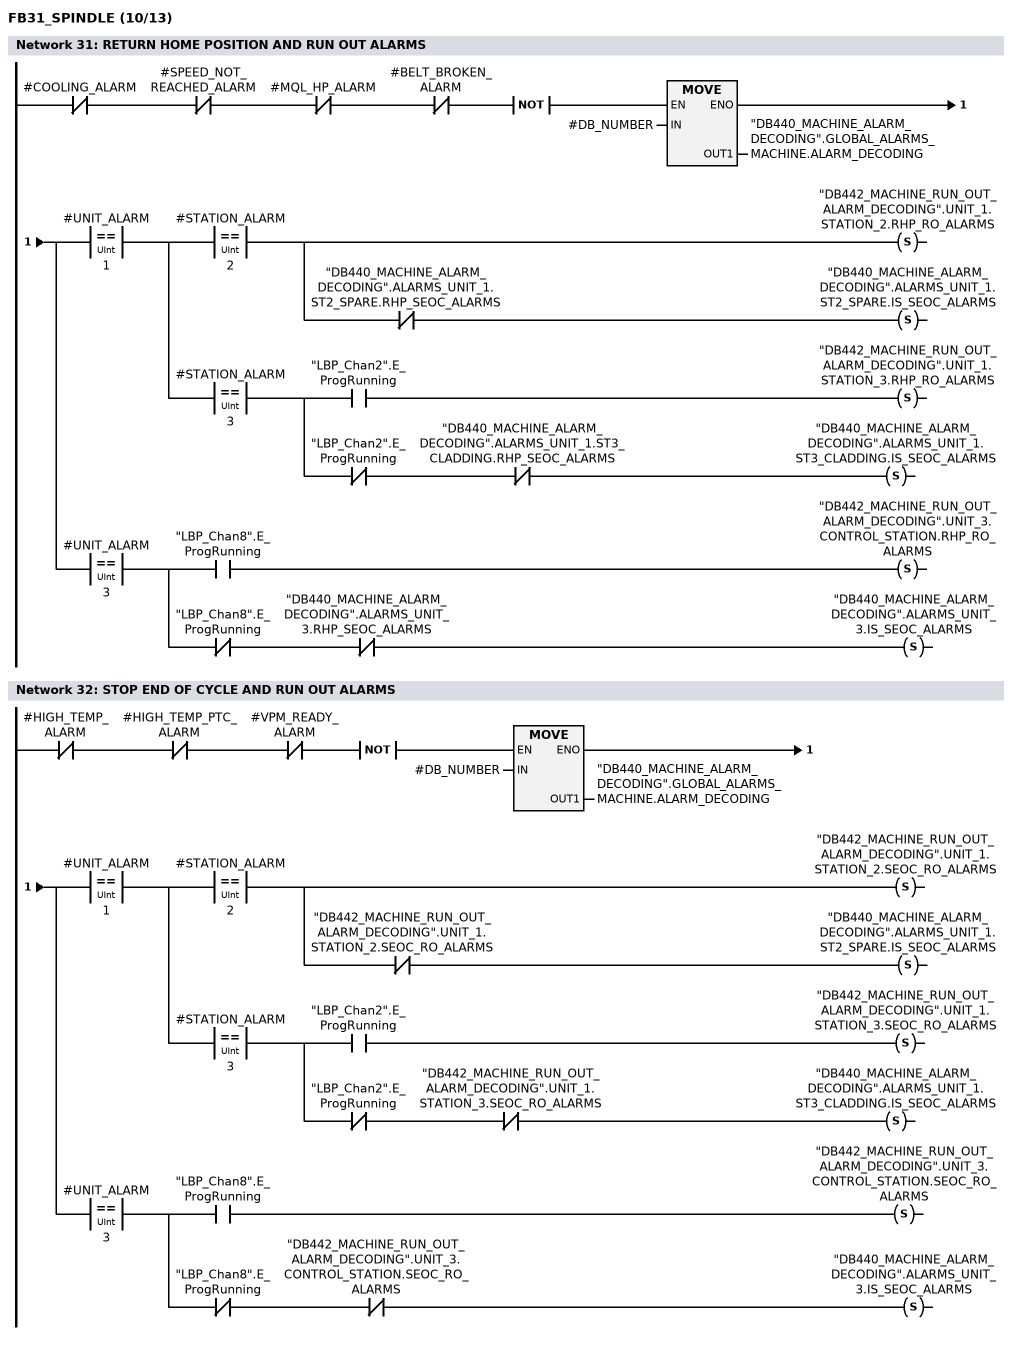
   RUNG wire#powerrail
      I_Contact( #COOLING_ALARM )
      I_Contact( #SPEED_NOT_REACHED_ALARM )
      I_Contact( #MQL_HP_ALARM )
      I_Contact( #BELT_BROKEN_ALARM )
      Not()
      Move(in := #DB_NUMBER, out1 => "DB440_MACHINE_ALARM_DECODING".GLOBAL_ALARMS_MACHINE.ALARM_DECODING)
      wire#w1
      { S7_Templates := "SrcType := UInt" } EQ_Contact(in1 := #UNIT_ALARM, in2 := 1)
      wire#w2
      { S7_Templates := "SrcType := UInt" } EQ_Contact(in1 := #STATION_ALARM, in2 := 2)
      wire#w3
      S_Coil( "DB442_MACHINE_RUN_OUT_ALARM_DECODING".UNIT_1.STATION_2.RHP_RO_ALARMS )
   END_RUNG
   RUNG wire#w3
      I_Contact( "DB440_MACHINE_ALARM_DECODING".ALARMS_UNIT_1.ST2_SPARE.RHP_SEOC_ALARMS )
      S_Coil( "DB440_MACHINE_ALARM_DECODING".ALARMS_UNIT_1.ST2_SPARE.IS_SEOC_ALARMS )
   END_RUNG
   RUNG wire#w2
      { S7_Templates := "SrcType := UInt" } EQ_Contact(in1 := #STATION_ALARM, in2 := 3)
      wire#w4
      Contact( "LBP_Chan2".E_ProgRunning )
      S_Coil( "DB442_MACHINE_RUN_OUT_ALARM_DECODING".UNIT_1.STATION_3.RHP_RO_ALARMS )
   END_RUNG
   RUNG wire#w4
      I_Contact( "LBP_Chan2".E_ProgRunning )
      I_Contact( "DB440_MACHINE_ALARM_DECODING".ALARMS_UNIT_1.ST3_CLADDING.RHP_SEOC_ALARMS )
      S_Coil( "DB440_MACHINE_ALARM_DECODING".ALARMS_UNIT_1.ST3_CLADDING.IS_SEOC_ALARMS )
   END_RUNG
   RUNG wire#w1
      { S7_Templates := "SrcType := UInt" } EQ_Contact(in1 := #UNIT_ALARM, in2 := 3)
      wire#w5
      Contact( "LBP_Chan8".E_ProgRunning )
      S_Coil( "DB442_MACHINE_RUN_OUT_ALARM_DECODING".UNIT_3.CONTROL_STATION.RHP_RO_ALARMS )
   END_RUNG
   RUNG wire#w5
      I_Contact( "LBP_Chan8".E_ProgRunning )
      I_Contact( "DB440_MACHINE_ALARM_DECODING".ALARMS_UNIT_3.RHP_SEOC_ALARMS )
      S_Coil( "DB440_MACHINE_ALARM_DECODING".ALARMS_UNIT_3.IS_SEOC_ALARMS )
   END_RUNG
   // the same network as SCL:
   #_w1 := NOT (NOT #COOLING_ALARM AND NOT #SPEED_NOT_REACHED_ALARM AND NOT #MQL_HP_ALARM AND NOT #BELT_BROKEN_ALARM);
   IF #_w1 THEN "DB440_MACHINE_ALARM_DECODING".GLOBAL_ALARMS_MACHINE.ALARM_DECODING := #DB_NUMBER; END_IF;
   #_w2 := #_w1 AND (#UNIT_ALARM = 1);
   #_w3 := #_w2 AND (#STATION_ALARM = 2);
   IF #_w3 THEN "DB442_MACHINE_RUN_OUT_ALARM_DECODING".UNIT_1.STATION_2.RHP_RO_ALARMS := TRUE; END_IF;
   IF #_w3 AND NOT "DB440_MACHINE_ALARM_DECODING".ALARMS_UNIT_1.ST2_SPARE.RHP_SEOC_ALARMS THEN
       "DB440_MACHINE_ALARM_DECODING".ALARMS_UNIT_1.ST2_SPARE.IS_SEOC_ALARMS := TRUE;
   END_IF;
   #_w4 := #_w2 AND (#STATION_ALARM = 3);
   IF #_w4 AND "LBP_Chan2".E_ProgRunning THEN
       "DB442_MACHINE_RUN_OUT_ALARM_DECODING".UNIT_1.STATION_3.RHP_RO_ALARMS := TRUE;
   END_IF;
   IF #_w4 AND NOT "LBP_Chan2".E_ProgRunning AND NOT "DB440_MACHINE_ALARM_DECODING".ALARMS_UNIT_1.ST3_CLADDING.RHP_SEOC_ALARMS THEN
       "DB440_MACHINE_ALARM_DECODING".ALARMS_UNIT_1.ST3_CLADDING.IS_SEOC_ALARMS := TRUE;
   END_IF;
   #_w5 := #_w1 AND (#UNIT_ALARM = 3);
   IF #_w5 AND "LBP_Chan8".E_ProgRunning THEN
       "DB442_MACHINE_RUN_OUT_ALARM_DECODING".UNIT_3.CONTROL_STATION.RHP_RO_ALARMS := TRUE;
   END_IF;
   IF #_w5 AND NOT "LBP_Chan8".E_ProgRunning AND NOT "DB440_MACHINE_ALARM_DECODING".ALARMS_UNIT_3.RHP_SEOC_ALARMS THEN
       "DB440_MACHINE_ALARM_DECODING".ALARMS_UNIT_3.IS_SEOC_ALARMS := TRUE;
   END_IF;
END_REGION

REGION Network 32: STOP END OF CYCLE AND RUN OUT ALARMS
   RUNG wire#powerrail
      I_Contact( #HIGH_TEMP_ALARM )
      I_Contact( #HIGH_TEMP_PTC_ALARM )
      I_Contact( #VPM_READY_ALARM )
      Not()
      { S7_GenerateENO := "TRUE" } Move(in := #DB_NUMBER, out1 => "DB440_MACHINE_ALARM_DECODING".GLOBAL_ALARMS_MACHINE.ALARM_DECODING)
      wire#w1
      { S7_Templates := "SrcType := UInt" } EQ_Contact(in1 := #UNIT_ALARM, in2 := 1)
      wire#w2
      { S7_Templates := "SrcType := UInt" } EQ_Contact(in1 := #STATION_ALARM, in2 := 2)
      wire#w3
      S_Coil( "DB442_MACHINE_RUN_OUT_ALARM_DECODING".UNIT_1.STATION_2.SEOC_RO_ALARMS )
   END_RUNG
   RUNG wire#w3
      I_Contact( "DB442_MACHINE_RUN_OUT_ALARM_DECODING".UNIT_1.STATION_2.SEOC_RO_ALARMS )
      S_Coil( "DB440_MACHINE_ALARM_DECODING".ALARMS_UNIT_1.ST2_SPARE.IS_SEOC_ALARMS )
   END_RUNG
   RUNG wire#w2
      { S7_Templates := "SrcType := UInt" } EQ_Contact(in1 := #STATION_ALARM, in2 := 3)
      wire#w4
      Contact( "LBP_Chan2".E_ProgRunning )
      S_Coil( "DB442_MACHINE_RUN_OUT_ALARM_DECODING".UNIT_1.STATION_3.SEOC_RO_ALARMS )
   END_RUNG
   RUNG wire#w4
      I_Contact( "LBP_Chan2".E_ProgRunning )
      I_Contact( "DB442_MACHINE_RUN_OUT_ALARM_DECODING".UNIT_1.STATION_3.SEOC_RO_ALARMS )
      S_Coil( "DB440_MACHINE_ALARM_DECODING".ALARMS_UNIT_1.ST3_CLADDING.IS_SEOC_ALARMS )
   END_RUNG
   RUNG wire#w1
      { S7_Templates := "SrcType := UInt" } EQ_Contact(in1 := #UNIT_ALARM, in2 := 3)
      wire#w5
      Contact( "LBP_Chan8".E_ProgRunning )
      S_Coil( "DB442_MACHINE_RUN_OUT_ALARM_DECODING".UNIT_3.CONTROL_STATION.SEOC_RO_ALARMS )
   END_RUNG
   RUNG wire#w5
      I_Contact( "LBP_Chan8".E_ProgRunning )
      I_Contact( "DB442_MACHINE_RUN_OUT_ALARM_DECODING".UNIT_3.CONTROL_STATION.SEOC_RO_ALARMS )
      S_Coil( "DB440_MACHINE_ALARM_DECODING".ALARMS_UNIT_3.IS_SEOC_ALARMS )
   END_RUNG
   // the same network as SCL:
   // ENO of a box is taken as its EN; it also drops when the box reports an error
   #_w1 := NOT (NOT #HIGH_TEMP_ALARM AND NOT #HIGH_TEMP_PTC_ALARM AND NOT #VPM_READY_ALARM);
   IF #_w1 THEN "DB440_MACHINE_ALARM_DECODING".GLOBAL_ALARMS_MACHINE.ALARM_DECODING := #DB_NUMBER; END_IF;
   #_w2 := #_w1 AND (#UNIT_ALARM = 1);
   #_w3 := #_w2 AND (#STATION_ALARM = 2);
   IF #_w3 THEN "DB442_MACHINE_RUN_OUT_ALARM_DECODING".UNIT_1.STATION_2.SEOC_RO_ALARMS := TRUE; END_IF;
   IF #_w3 AND NOT "DB442_MACHINE_RUN_OUT_ALARM_DECODING".UNIT_1.STATION_2.SEOC_RO_ALARMS THEN
       "DB440_MACHINE_ALARM_DECODING".ALARMS_UNIT_1.ST2_SPARE.IS_SEOC_ALARMS := TRUE;
   END_IF;
   #_w4 := #_w2 AND (#STATION_ALARM = 3);
   IF #_w4 AND "LBP_Chan2".E_ProgRunning THEN
       "DB442_MACHINE_RUN_OUT_ALARM_DECODING".UNIT_1.STATION_3.SEOC_RO_ALARMS := TRUE;
   END_IF;
   IF #_w4 AND NOT "LBP_Chan2".E_ProgRunning AND NOT "DB442_MACHINE_RUN_OUT_ALARM_DECODING".UNIT_1.STATION_3.SEOC_RO_ALARMS THEN
       "DB440_MACHINE_ALARM_DECODING".ALARMS_UNIT_1.ST3_CLADDING.IS_SEOC_ALARMS := TRUE;
   END_IF;
   #_w5 := #_w1 AND (#UNIT_ALARM = 3);
   IF #_w5 AND "LBP_Chan8".E_ProgRunning THEN
       "DB442_MACHINE_RUN_OUT_ALARM_DECODING".UNIT_3.CONTROL_STATION.SEOC_RO_ALARMS := TRUE;
   END_IF;
   IF #_w5 AND NOT "LBP_Chan8".E_ProgRunning AND NOT "DB442_MACHINE_RUN_OUT_ALARM_DECODING".UNIT_3.CONTROL_STATION.SEOC_RO_ALARMS THEN
       "DB440_MACHINE_ALARM_DECODING".ALARMS_UNIT_3.IS_SEOC_ALARMS := TRUE;
   END_IF;
END_REGION

REGION Network 33: PROGRESSIVE STOP POWDER ALARMS
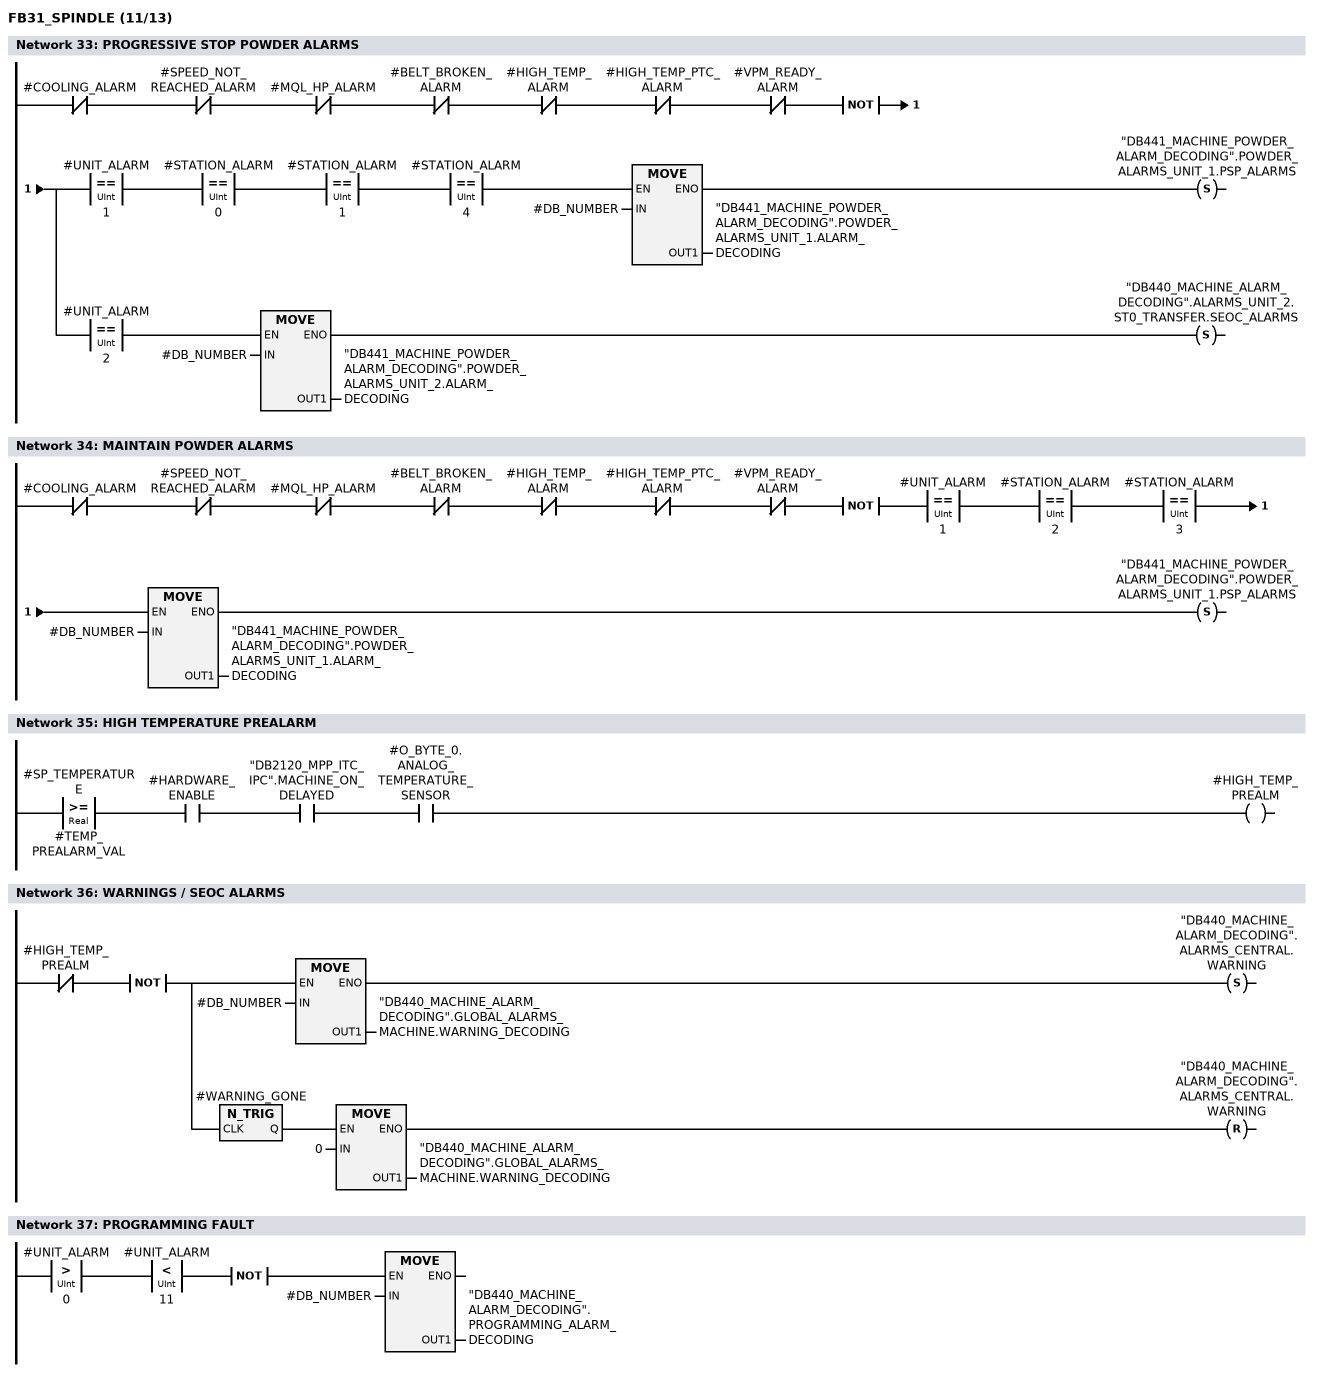
   RUNG wire#powerrail
      I_Contact( #COOLING_ALARM )
      I_Contact( #SPEED_NOT_REACHED_ALARM )
      I_Contact( #MQL_HP_ALARM )
      I_Contact( #BELT_BROKEN_ALARM )
      I_Contact( #HIGH_TEMP_ALARM )
      I_Contact( #HIGH_TEMP_PTC_ALARM )
      I_Contact( #VPM_READY_ALARM )
      Not()
      wire#w1
      { S7_Templates := "SrcType := UInt" } EQ_Contact(in1 := #UNIT_ALARM, in2 := 1)
      { S7_Templates := "SrcType := UInt" } EQ_Contact(in1 := #STATION_ALARM, in2 := 0)
      { S7_Templates := "SrcType := UInt" } EQ_Contact(in1 := #STATION_ALARM, in2 := 1)
      { S7_Templates := "SrcType := UInt" } EQ_Contact(in1 := #STATION_ALARM, in2 := 4)
      { S7_GenerateENO := "TRUE" } Move(in := #DB_NUMBER, out1 => "DB441_MACHINE_POWDER_ALARM_DECODING".POWDER_ALARMS_UNIT_1.ALARM_DECODING)
      S_Coil( "DB441_MACHINE_POWDER_ALARM_DECODING".POWDER_ALARMS_UNIT_1.PSP_ALARMS )
   END_RUNG
   RUNG wire#w1
      { S7_Templates := "SrcType := UInt" } EQ_Contact(in1 := #UNIT_ALARM, in2 := 2)
      { S7_GenerateENO := "TRUE" } Move(in := #DB_NUMBER, out1 => "DB441_MACHINE_POWDER_ALARM_DECODING".POWDER_ALARMS_UNIT_2.ALARM_DECODING)
      S_Coil( "DB440_MACHINE_ALARM_DECODING".ALARMS_UNIT_2.ST0_TRANSFER.SEOC_ALARMS )
   END_RUNG
   // the same network as SCL:
   // ENO of a box is taken as its EN; it also drops when the box reports an error
   #_w1 := NOT (NOT #COOLING_ALARM AND NOT #SPEED_NOT_REACHED_ALARM AND NOT #MQL_HP_ALARM AND NOT #BELT_BROKEN_ALARM AND NOT #HIGH_TEMP_ALARM AND NOT #HIGH_TEMP_PTC_ALARM AND NOT #VPM_READY_ALARM);
   IF #_w1 AND (#UNIT_ALARM = 1) AND (#STATION_ALARM = 0) AND (#STATION_ALARM = 1) AND (#STATION_ALARM = 4) THEN
       "DB441_MACHINE_POWDER_ALARM_DECODING".POWDER_ALARMS_UNIT_1.ALARM_DECODING := #DB_NUMBER;
       "DB441_MACHINE_POWDER_ALARM_DECODING".POWDER_ALARMS_UNIT_1.PSP_ALARMS := TRUE;
   END_IF;
   IF #_w1 AND (#UNIT_ALARM = 2) THEN
       "DB441_MACHINE_POWDER_ALARM_DECODING".POWDER_ALARMS_UNIT_2.ALARM_DECODING := #DB_NUMBER;
       "DB440_MACHINE_ALARM_DECODING".ALARMS_UNIT_2.ST0_TRANSFER.SEOC_ALARMS := TRUE;
   END_IF;
END_REGION

REGION Network 34: MAINTAIN POWDER ALARMS
   RUNG wire#powerrail
      I_Contact( #COOLING_ALARM )
      I_Contact( #SPEED_NOT_REACHED_ALARM )
      I_Contact( #MQL_HP_ALARM )
      I_Contact( #BELT_BROKEN_ALARM )
      I_Contact( #HIGH_TEMP_ALARM )
      I_Contact( #HIGH_TEMP_PTC_ALARM )
      I_Contact( #VPM_READY_ALARM )
      Not()
      { S7_Templates := "SrcType := UInt" } EQ_Contact(in1 := #UNIT_ALARM, in2 := 1)
      { S7_Templates := "SrcType := UInt" } EQ_Contact(in1 := #STATION_ALARM, in2 := 2)
      { S7_Templates := "SrcType := UInt" } EQ_Contact(in1 := #STATION_ALARM, in2 := 3)
      { S7_GenerateENO := "TRUE" } Move(in := #DB_NUMBER, out1 => "DB441_MACHINE_POWDER_ALARM_DECODING".POWDER_ALARMS_UNIT_1.ALARM_DECODING)
      S_Coil( "DB441_MACHINE_POWDER_ALARM_DECODING".POWDER_ALARMS_UNIT_1.PSP_ALARMS )
   END_RUNG
   // the same network as SCL:
   // ENO of a box is taken as its EN; it also drops when the box reports an error
   IF NOT (NOT #COOLING_ALARM AND NOT #SPEED_NOT_REACHED_ALARM AND NOT #MQL_HP_ALARM AND NOT #BELT_BROKEN_ALARM AND NOT #HIGH_TEMP_ALARM AND NOT #HIGH_TEMP_PTC_ALARM AND NOT #VPM_READY_ALARM) AND (#UNIT_ALARM = 1) AND (#STATION_ALARM = 2) AND (#STATION_ALARM = 3) THEN
       "DB441_MACHINE_POWDER_ALARM_DECODING".POWDER_ALARMS_UNIT_1.ALARM_DECODING := #DB_NUMBER;
       "DB441_MACHINE_POWDER_ALARM_DECODING".POWDER_ALARMS_UNIT_1.PSP_ALARMS := TRUE;
   END_IF;
END_REGION

REGION Network 35: HIGH TEMPERATURE PREALARM
   RUNG wire#powerrail
      { S7_Templates := "SrcType := Real" } GE_Contact(in1 := #SP_TEMPERATURE, in2 := #TEMP_PREALARM_VAL)
      Contact( #HARDWARE_ENABLE )
      Contact( "DB2120_MPP_ITC_IPC".MACHINE_ON_DELAYED )
      Contact( #O_BYTE_0.ANALOG_TEMPERATURE_SENSOR )
      Coil( #HIGH_TEMP_PREALM )
   END_RUNG
   // the same network as SCL:
   #HIGH_TEMP_PREALM := (#SP_TEMPERATURE >= #TEMP_PREALARM_VAL) AND #HARDWARE_ENABLE AND "DB2120_MPP_ITC_IPC".MACHINE_ON_DELAYED AND #O_BYTE_0.ANALOG_TEMPERATURE_SENSOR;
END_REGION

REGION Network 36: WARNINGS / SEOC ALARMS
   RUNG wire#powerrail
      I_Contact( #HIGH_TEMP_PREALM )
      Not()
      wire#w1
      { S7_GenerateENO := "TRUE" } Move(in := #DB_NUMBER, out1 => "DB440_MACHINE_ALARM_DECODING".GLOBAL_ALARMS_MACHINE.WARNING_DECODING)
      S_Coil( "DB440_MACHINE_ALARM_DECODING".ALARMS_CENTRAL.WARNING )
   END_RUNG
   RUNG wire#w1
      N_Trig( #WARNING_GONE )
      { S7_GenerateENO := "TRUE" } Move(in := 0, out1 => "DB440_MACHINE_ALARM_DECODING".GLOBAL_ALARMS_MACHINE.WARNING_DECODING)
      R_Coil( "DB440_MACHINE_ALARM_DECODING".ALARMS_CENTRAL.WARNING )
   END_RUNG
   // the same network as SCL:
   // ENO of a box is taken as its EN; it also drops when the box reports an error
   #_w1 := NOT (NOT #HIGH_TEMP_PREALM);
   IF #_w1 THEN
       "DB440_MACHINE_ALARM_DECODING".GLOBAL_ALARMS_MACHINE.WARNING_DECODING := #DB_NUMBER;
       "DB440_MACHINE_ALARM_DECODING".ALARMS_CENTRAL.WARNING := TRUE;
   END_IF;
   #_w2 := NOT #_w1 AND #WARNING_GONE;   // falling edge
   #WARNING_GONE := #_w1;
   IF #_w2 THEN
       "DB440_MACHINE_ALARM_DECODING".GLOBAL_ALARMS_MACHINE.WARNING_DECODING := 0;
       "DB440_MACHINE_ALARM_DECODING".ALARMS_CENTRAL.WARNING := FALSE;
   END_IF;
END_REGION

REGION Network 37: PROGRAMMING FAULT
   RUNG wire#powerrail
      { S7_Templates := "SrcType := UInt" } GT_Contact(in1 := #UNIT_ALARM, in2 := 0)
      { S7_Templates := "SrcType := UInt" } LT_Contact(in1 := #UNIT_ALARM, in2 := 11)
      Not()
      Move(in := #DB_NUMBER, out1 => "DB440_MACHINE_ALARM_DECODING".PROGRAMMING_ALARM_DECODING)
   END_RUNG
   // the same network as SCL:
   IF NOT ((#UNIT_ALARM > 0) AND (#UNIT_ALARM < 11)) THEN
       "DB440_MACHINE_ALARM_DECODING".PROGRAMMING_ALARM_DECODING := #DB_NUMBER;
   END_IF;
END_REGION

REGION Network 38: OPERATOR HELP / HELP
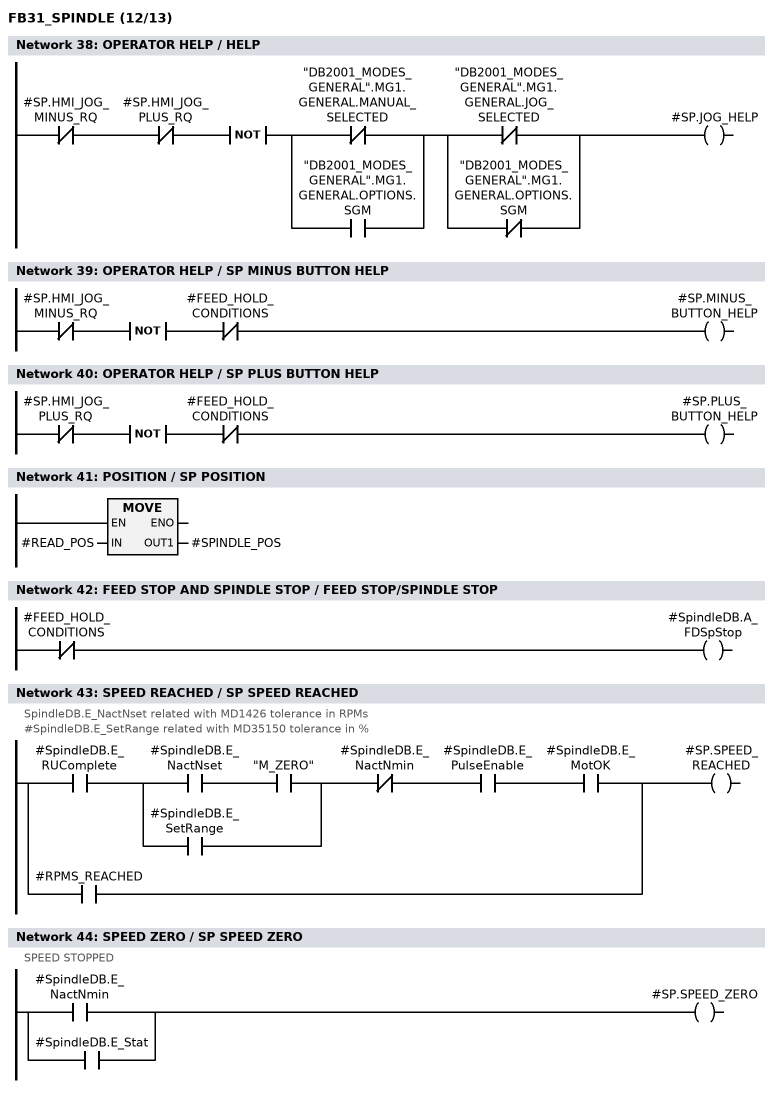
   RUNG wire#powerrail
      I_Contact( #SP.HMI_JOG_MINUS_RQ )
      I_Contact( #SP.HMI_JOG_PLUS_RQ )
      Not()
      wire#w1
      I_Contact( "DB2001_MODES_GENERAL".MG1.GENERAL.MANUAL_SELECTED )
      wire#w2
      I_Contact( "DB2001_MODES_GENERAL".MG1.GENERAL.JOG_SELECTED )
      wire#w3
      Coil( #SP.JOG_HELP )
   END_RUNG
   RUNG wire#w1
      Contact( "DB2001_MODES_GENERAL".MG1.GENERAL.OPTIONS.SGM )
   END_RUNG wire#w2
   RUNG wire#w2
      I_Contact( "DB2001_MODES_GENERAL".MG1.GENERAL.OPTIONS.SGM )
   END_RUNG wire#w3
   // the same network as SCL:
   #SP.JOG_HELP := NOT (NOT #SP.HMI_JOG_MINUS_RQ AND NOT #SP.HMI_JOG_PLUS_RQ) AND (NOT "DB2001_MODES_GENERAL".MG1.GENERAL.MANUAL_SELECTED OR "DB2001_MODES_GENERAL".MG1.GENERAL.OPTIONS.SGM) AND (NOT "DB2001_MODES_GENERAL".MG1.GENERAL.JOG_SELECTED OR NOT "DB2001_MODES_GENERAL".MG1.GENERAL.OPTIONS.SGM);
END_REGION

REGION Network 39: OPERATOR HELP / SP MINUS BUTTON HELP
   RUNG wire#powerrail
      I_Contact( #SP.HMI_JOG_MINUS_RQ )
      Not()
      I_Contact( #FEED_HOLD_CONDITIONS )
      Coil( #SP.MINUS_BUTTON_HELP )
   END_RUNG
   // the same network as SCL:
   #SP.MINUS_BUTTON_HELP := NOT (NOT #SP.HMI_JOG_MINUS_RQ) AND NOT #FEED_HOLD_CONDITIONS;
END_REGION

REGION Network 40: OPERATOR HELP / SP PLUS BUTTON HELP
   RUNG wire#powerrail
      I_Contact( #SP.HMI_JOG_PLUS_RQ )
      Not()
      I_Contact( #FEED_HOLD_CONDITIONS )
      Coil( #SP.PLUS_BUTTON_HELP )
   END_RUNG
   // the same network as SCL:
   #SP.PLUS_BUTTON_HELP := NOT (NOT #SP.HMI_JOG_PLUS_RQ) AND NOT #FEED_HOLD_CONDITIONS;
END_REGION

REGION Network 41: POSITION / SP POSITION
   RUNG wire#powerrail
      { S7_GenerateENO := "TRUE" } Move(in := #READ_POS, out1 => #SPINDLE_POS)
   END_RUNG
   // the same network as SCL:
   #SPINDLE_POS := #READ_POS;
END_REGION

REGION Network 42: FEED STOP AND SPINDLE STOP / FEED STOP/SPINDLE STOP
   RUNG wire#powerrail
      I_Contact( #FEED_HOLD_CONDITIONS )
      Coil( #SpindleDB.A_FDSpStop )
   END_RUNG
   // the same network as SCL:
   #SpindleDB.A_FDSpStop := NOT #FEED_HOLD_CONDITIONS;
END_REGION

REGION Network 43: SPEED REACHED / SP SPEED REACHED
   // SpindleDB.E_NactNset related with MD1426 tolerance in RPMs
   // #SpindleDB.E_SetRange related with MD35150 tolerance in %
   RUNG wire#powerrail
      Contact( #SpindleDB.E_RUComplete )
      wire#w1
      Contact( #SpindleDB.E_NactNset )
      Contact( "M_ZERO" )
      wire#w2
      I_Contact( #SpindleDB.E_NactNmin )
      Contact( #SpindleDB.E_PulseEnable )
      Contact( #SpindleDB.E_MotOK )
      wire#w3
      Coil( #SP.SPEED_REACHED )
   END_RUNG
   RUNG wire#w1
      Contact( #SpindleDB.E_SetRange )
   END_RUNG wire#w2
   RUNG wire#powerrail
      Contact( #RPMS_REACHED )
   END_RUNG wire#w3
   // the same network as SCL:
   #SP.SPEED_REACHED := (#SpindleDB.E_RUComplete AND ((#SpindleDB.E_NactNset AND "M_ZERO") OR #SpindleDB.E_SetRange) AND NOT #SpindleDB.E_NactNmin AND #SpindleDB.E_PulseEnable AND #SpindleDB.E_MotOK) OR #RPMS_REACHED;
END_REGION

REGION Network 44: SPEED ZERO / SP SPEED ZERO
   // SPEED STOPPED
   RUNG wire#powerrail
      Contact( #SpindleDB.E_NactNmin )
      wire#w1
      Coil( #SP.SPEED_ZERO )
   END_RUNG
   RUNG wire#powerrail
      Contact( #SpindleDB.E_Stat )
   END_RUNG wire#w1
   // the same network as SCL:
   #SP.SPEED_ZERO := #SpindleDB.E_NactNmin OR #SpindleDB.E_Stat;
END_REGION

REGION Network 45: CALL FB33 SAFETY POSITIONS
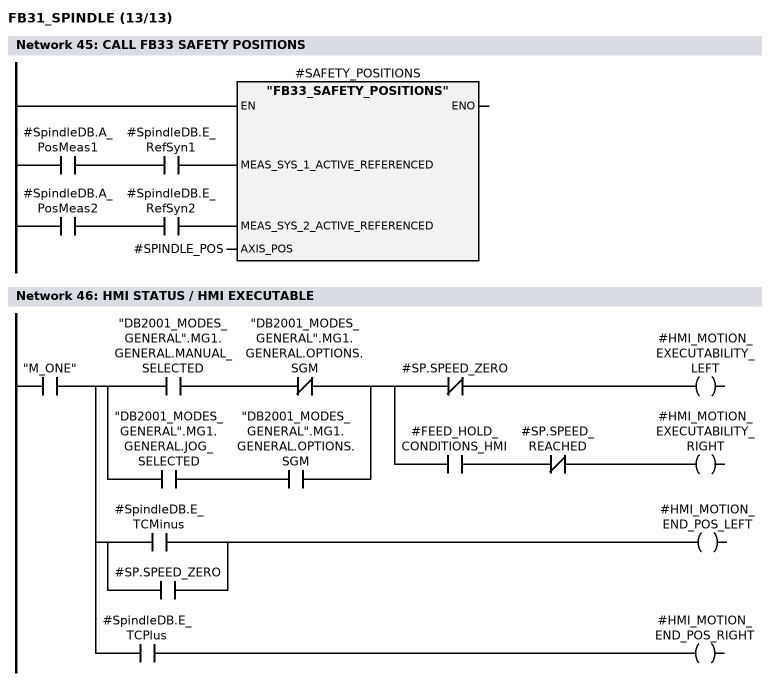
   RUNG wire#powerrail
      #SAFETY_POSITIONS(MEAS_SYS_1_ACTIVE_REFERENCED := wire#w1, MEAS_SYS_2_ACTIVE_REFERENCED := wire#w2, AXIS_POS := #SPINDLE_POS)
   END_RUNG
   RUNG wire#powerrail
      Contact( #SpindleDB.A_PosMeas1 )
      Contact( #SpindleDB.E_RefSyn1 )
   END_RUNG wire#w1
   RUNG wire#powerrail
      Contact( #SpindleDB.A_PosMeas2 )
      Contact( #SpindleDB.E_RefSyn2 )
   END_RUNG wire#w2
   // the same network as SCL:
   #SAFETY_POSITIONS(MEAS_SYS_1_ACTIVE_REFERENCED := #SpindleDB.A_PosMeas1 AND #SpindleDB.E_RefSyn1,   // "FB33_SAFETY_POSITIONS"
                     MEAS_SYS_2_ACTIVE_REFERENCED := #SpindleDB.A_PosMeas2 AND #SpindleDB.E_RefSyn2,
                     AXIS_POS := #SPINDLE_POS);
END_REGION

REGION Network 46: HMI STATUS / HMI EXECUTABLE
   RUNG wire#powerrail
      Contact( "M_ONE" )
      wire#w1
      Contact( "DB2001_MODES_GENERAL".MG1.GENERAL.MANUAL_SELECTED )
      I_Contact( "DB2001_MODES_GENERAL".MG1.GENERAL.OPTIONS.SGM )
      wire#w2
      I_Contact( #SP.SPEED_ZERO )
      Coil( #HMI_MOTION_EXECUTABILITY_LEFT )
   END_RUNG
   RUNG wire#w1
      Contact( "DB2001_MODES_GENERAL".MG1.GENERAL.JOG_SELECTED )
      Contact( "DB2001_MODES_GENERAL".MG1.GENERAL.OPTIONS.SGM )
   END_RUNG wire#w2
   RUNG wire#w2
      Contact( #FEED_HOLD_CONDITIONS_HMI )
      I_Contact( #SP.SPEED_REACHED )
      Coil( #HMI_MOTION_EXECUTABILITY_RIGHT )
   END_RUNG
   RUNG wire#w1
      Contact( #SpindleDB.E_TCMinus )
      wire#w3
      Coil( #HMI_MOTION_END_POS_LEFT )
   END_RUNG
   RUNG wire#w1
      Contact( #SP.SPEED_ZERO )
   END_RUNG wire#w3
   RUNG wire#w1
      Contact( #SpindleDB.E_TCPlus )
      Coil( #HMI_MOTION_END_POS_RIGHT )
   END_RUNG
   // the same network as SCL:
   #_w1 := "M_ONE" AND (("DB2001_MODES_GENERAL".MG1.GENERAL.MANUAL_SELECTED AND NOT "DB2001_MODES_GENERAL".MG1.GENERAL.OPTIONS.SGM) OR ("DB2001_MODES_GENERAL".MG1.GENERAL.JOG_SELECTED AND "DB2001_MODES_GENERAL".MG1.GENERAL.OPTIONS.SGM));
   #HMI_MOTION_EXECUTABILITY_LEFT := #_w1 AND NOT #SP.SPEED_ZERO;
   #HMI_MOTION_EXECUTABILITY_RIGHT := #_w1 AND #FEED_HOLD_CONDITIONS_HMI AND NOT #SP.SPEED_REACHED;
   #HMI_MOTION_END_POS_LEFT := "M_ONE" AND (#SpindleDB.E_TCMinus OR #SP.SPEED_ZERO);
   #HMI_MOTION_END_POS_RIGHT := "M_ONE" AND #SpindleDB.E_TCPlus;
END_REGION
END_FUNCTION_BLOCK
